KUKA KRL program: EPS_2_25362_MH2A_A_20251103083054.src

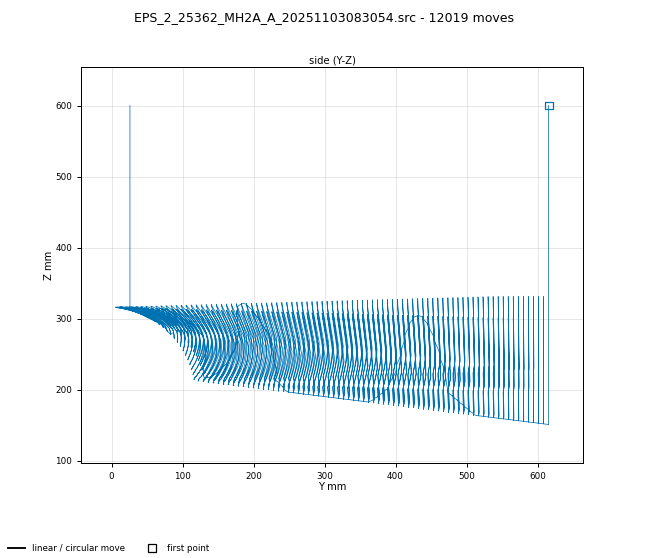
[picture p0: tool path of EPS_2_25362_MH2A_A_20251103083054.src, 12019 of 12021 moves have a stored position in this frame; points joined in program order, loops and branches not executed]
&ACCESS RVP
&REL 4
&COMMENT QRS 19112012
&PARAM EDITMASK = *
DEF PART()
EXT BAS (BAS_COMMAND :IN,REAL :IN )
INT I
BAS (#INITMOV,0 )

;KUKA QRS Post kuka4.cps  Date:22-06-2017 !

File_ID=2899

QRS_PRE_INIT()

;Init var - Until changes are made in qrs_pre_init
Outlet_Square_prg=0
Inlet_1_Square_prg=0
Inlet_2_Square_prg=0
Inlet_3_Square_prg=0
Inlet_4_Square_prg=0
Inlet_5_Square_prg=0

Outlet_1={X 0.000, Y 537.380, Z 230.500, B 0.000, E1 0.000 }
Inlet_1={X 0.000, Y 539.550, Z 200.500, B 0.000, E1 178.000 }
Outlet_1_type=201
Inlet_1_type=201
;QRS#1=Sidecore dimensions
;QRS#2=200-8" PVC SDR 35
;QRS#3=200-8" PVC SDR 35
;QRS#4=
;QRS#5=
;QRS#6=
;QRS#7=
;QRS#8=
;QRS#9=12-08 PSX
;QRS#10=12-08 PSX
;QRS#11=
;QRS#12=
;QRS#13=
;QRS#14=
;QRS#15=
;QRS#16=1220x127x610 2'
;QRS#17=EPS Height
;QRS#18=331
;QRS#19=*
;QRS#20= UPDATED VERSION 22-06-2017
;QRS#21=*
Outlet_Square=0100
Inlet_1_Square=0100
Inlet_2_Square=0
Inlet_3_Square=0
Inlet_4_Square=0
Inlet_5_Square=0
Mill_Square=1
Outlet_Square_Prg=204
Inlet_1_Square_prg=204

QRS_INIT()

$ADVANCE=5

; T1
PTP {E1 173.58,E2 173.58}
PTP {X 0,Y 615.495,A -85,B 0,C 180,E1 173.58,E2 173.58,E3 0,E4 0,E5 0,E6 0}
QRS_SPEED_INIT()
LIN {X 0,Y 615.495,Z 600,A -85,B 0,C 180,E1 173.58,E2 173.58,E3 0,E4 0,E5 0,E6 0} C_VEL
LIN {X 0,Y 615.495,Z 160.868,A -85,B 0,C 180,E1 173.58,E2 173.58} C_VEL
LIN {X 0,Y 615.495,Z 152.689,A -85,B 0,C 180,E1 173.58,E2 173.58} C_VEL
LIN {X 0,Y 615.483,Z 150.689,A -85,B 0,C 180,E1 173.393,E2 173.393} C_VEL
LIN {X 0,Y 615.483,Z 150.7,A -85,B 0,C 180,E1 170.801,E2 170.801} C_VEL
LIN {X 0,Y 615.439,Z 150.7,A -85,B 0,C 180,E1 168.138,E2 168.138} C_VEL
LIN {X 0,Y 615.491,Z 150.691,A -85,B 0,C 180,E1 165.451,E2 165.451} C_VEL
LIN {X 0,Y 615.482,Z 150.697,A -85,B 0,C 180,E1 162.729,E2 162.729} C_VEL
LIN {X 0,Y 615.477,Z 150.69,A -85,B 0,C 180,E1 159.967,E2 159.967} C_VEL
LIN {X 0,Y 615.463,Z 150.7,A -85,B 0,C 180,E1 157.154,E2 157.154} C_VEL
LIN {X 0,Y 615.457,Z 150.7,A -85,B 0,C 180,E1 154.43,E2 154.43} C_VEL
LIN {X 0,Y 615.47,Z 150.692,A -85,B 0,C 180,E1 151.546,E2 151.546} C_VEL
LIN {X 0,Y 615.484,Z 150.7,A -85,B 0,C 180,E1 148.909,E2 148.909} C_VEL
LIN {X 0,Y 615.472,Z 150.692,A -85,B 0,C 180,E1 146.463,E2 146.463} C_VEL
LIN {X 0,Y 615.451,Z 150.7,A -85,B 0,C 180,E1 143.572,E2 143.572} C_VEL
LIN {X 0,Y 615.462,Z 150.7,A -85,B 0,C 180,E1 140.936,E2 140.936} C_VEL
LIN {X 0,Y 615.493,Z 150.691,A -85,B 0,C 180,E1 138.526,E2 138.526} C_VEL
LIN {X 0,Y 615.483,Z 150.696,A -85,B 0,C 180,E1 135.849,E2 135.849} C_VEL
LIN {X 0,Y 615.463,Z 150.693,A -85,B 0,C 180,E1 133.044,E2 133.044} C_VEL
LIN {X 0,Y 615.491,Z 150.7,A -85,B 0,C 180,E1 130.603,E2 130.603} C_VEL
LIN {X 0,Y 615.445,Z 150.698,A -85,B 0,C 180,E1 128.006,E2 128.006} C_VEL
LIN {X 0,Y 615.489,Z 150.883,A -85,B 0,C 180,E1 127.239,E2 127.239} C_VEL
LIN {X 0,Y 615.484,Z 155.327,A -85,B 0,C 180,E1 124.699,E2 124.699} C_VEL
LIN {X 0,Y 615.462,Z 159.55,A -85,B 0,C 180,E1 122.326,E2 122.326} C_VEL
LIN {X 0,Y 615.495,Z 164.12,A -85,B 0,C 180,E1 119.795,E2 119.795} C_VEL
LIN {X 0,Y 615.496,Z 169.29,A -85,B 0,C 180,E1 117.045,E2 117.045} C_VEL
LIN {X 0,Y 615.488,Z 174.63,A -85,B 0,C 180,E1 114.271,E2 114.271} C_VEL
LIN {X 0,Y 615.486,Z 180.203,A -85,B 0,C 180,E1 111.431,E2 111.431} C_VEL
LIN {X 0,Y 615.475,Z 185.852,A -85,B 0,C 180,E1 108.6,E2 108.6} C_VEL
LIN {X 0,Y 615.458,Z 191.315,A -85,B 0,C 180,E1 105.905,E2 105.905} C_VEL
LIN {X 0,Y 615.497,Z 196.111,A -85,B 0,C 180,E1 103.558,E2 103.558} C_VEL
LIN {X 0,Y 615.486,Z 208.924,A -85,B 0,C 180,E1 103.285,E2 103.285} C_VEL
LIN {X 0,Y 615.445,Z 222.003,A -85,B 0,C 180,E1 102.866,E2 102.866} C_VEL
LIN {X 0,Y 615.432,Z 233.538,A -85,B 0,C 180,E1 102.363,E2 102.363} C_VEL
LIN {X 0,Y 615.477,Z 244.06,A -85,B 0,C 180,E1 101.777,E2 101.777} C_VEL
LIN {X 0,Y 615.496,Z 254.612,A -85,B 0,C 180,E1 101.041,E2 101.041} C_VEL
LIN {X 0,Y 615.498,Z 264.458,A -85,B 0,C 180,E1 100.194,E2 100.194} C_VEL
LIN {X 0,Y 615.496,Z 272.355,A -85,B 0,C 180,E1 99.364,E2 99.364} C_VEL
LIN {X 0,Y 615.497,Z 280.04,A -85,B 0,C 180,E1 98.371,E2 98.371} C_VEL
LIN {X 0,Y 615.495,Z 287.099,A -85,B 0,C 180,E1 97.215,E2 97.215} C_VEL
LIN {X 0,Y 615.496,Z 291.782,A -85,B 0,C 180,E1 96.227,E2 96.227} C_VEL
LIN {X 0,Y 615.498,Z 295.355,A -85,B 0,C 180,E1 95.241,E2 95.241} C_VEL
LIN {X 0,Y 615.496,Z 297.203,A -85,B 0,C 180,E1 94.585,E2 94.585} C_VEL
LIN {X 0,Y 615.497,Z 298.591,A -85,B 0,C 180,E1 93.929,E2 93.929} C_VEL
LIN {X 0,Y 615.495,Z 300.167,A -85,B 0,C 180,E1 92.618,E2 92.618} C_VEL
LIN {X 0,Y 615.5,Z 300.387,A -85,B 0,C 180,E1 91.963,E2 91.963} C_VEL
LIN {X 0,Y 615.495,Z 299.59,A -85,B 0,C 180,E1 90.655,E2 90.655} C_VEL
LIN {X 0,Y 615.497,Z 298.622,A -85,B 0,C 180,E1 90,E2 90} C_VEL
LIN {X 0,Y 615.494,Z 297.256,A -85,B 0,C 180,E1 89.346,E2 89.346} C_VEL
LIN {X 0,Y 615.496,Z 294.383,A -85,B 0,C 180,E1 88.365,E2 88.365} C_VEL
LIN {X 0,Y 615.498,Z 290.494,A -85,B 0,C 180,E1 87.383,E2 87.383} C_VEL
LIN {X 0,Y 615.496,Z 285.486,A -85,B 0,C 180,E1 86.4,E2 86.4} C_VEL
LIN {X 0,Y 615.498,Z 279.198,A -85,B 0,C 180,E1 85.416,E2 85.416} C_VEL
LIN {X 0,Y 615.498,Z 271.326,A -85,B 0,C 180,E1 84.431,E2 84.431} C_VEL
LIN {X 0,Y 615.498,Z 261.549,A -85,B 0,C 180,E1 83.444,E2 83.444} C_VEL
LIN {X 0,Y 615.499,Z 251.282,A -85,B 0,C 180,E1 82.621,E2 82.621} C_VEL
LIN {X 0,Y 615.454,Z 239.751,A -85,B 0,C 180,E1 81.877,E2 81.877} C_VEL
LIN {X 0,Y 615.435,Z 228.231,A -85,B 0,C 180,E1 81.298,E2 81.298} C_VEL
LIN {X 0,Y 615.465,Z 216.308,A -85,B 0,C 180,E1 80.843,E2 80.843} C_VEL
LIN {X 0,Y 615.499,Z 204.261,A -85,B 0,C 180,E1 80.512,E2 80.512} C_VEL
LIN {X 0,Y 615.487,Z 196.102,A -85,B 0,C 180,E1 80.346,E2 80.346} C_VEL
LIN {X 0,Y 615.472,Z 191.59,A -85,B 0,C 180,E1 78.14,E2 78.14} C_VEL
LIN {X 0,Y 615.467,Z 186.138,A -85,B 0,C 180,E1 75.452,E2 75.452} C_VEL
LIN {X 0,Y 615.492,Z 180.706,A -85,B 0,C 180,E1 72.731,E2 72.731} C_VEL
LIN {X 0,Y 615.478,Z 175.27,A -85,B 0,C 180,E1 69.969,E2 69.969} C_VEL
LIN {X 0,Y 615.477,Z 169.856,A -85,B 0,C 180,E1 67.157,E2 67.157} C_VEL
LIN {X 0,Y 615.493,Z 164.438,A -85,B 0,C 180,E1 64.287,E2 64.287} C_VEL
LIN {X 0,Y 615.46,Z 159.498,A -85,B 0,C 180,E1 61.556,E2 61.556} C_VEL
LIN {X 0,Y 615.49,Z 154.803,A -85,B 0,C 180,E1 58.915,E2 58.915} C_VEL
LIN {X 0,Y 615.466,Z 150.699,A -85,B 0,C 180,E1 56.47,E2 56.47} C_VEL
LIN {X 0,Y 615.43,Z 150.7,A -85,B 0,C 180,E1 54.175,E2 54.175} C_VEL
LIN {X 0,Y 615.45,Z 150.7,A -85,B 0,C 180,E1 51.933,E2 51.933} C_VEL
LIN {X 0,Y 615.489,Z 150.692,A -85,B 0,C 180,E1 49.398,E2 49.398} C_VEL
LIN {X 0,Y 615.471,Z 150.694,A -85,B 0,C 180,E1 46.758,E2 46.758} C_VEL
LIN {X 0,Y 615.477,Z 150.692,A -85,B 0,C 180,E1 44.001,E2 44.001} C_VEL
LIN {X 0,Y 615.489,Z 150.701,A -85,B 0,C 180,E1 41.1,E2 41.1} C_VEL
LIN {X 0,Y 615.453,Z 150.699,A -85,B 0,C 180,E1 38.907,E2 38.907} C_VEL
LIN {X 0,Y 615.436,Z 150.7,A -85,B 0,C 180,E1 36.429,E2 36.429} C_VEL
LIN {X 0,Y 615.463,Z 150.695,A -85,B 0,C 180,E1 33.538,E2 33.538} C_VEL
LIN {X 0,Y 615.469,Z 150.697,A -85,B 0,C 180,E1 30.921,E2 30.921} C_VEL
LIN {X 0,Y 615.485,Z 150.692,A -85,B 0,C 180,E1 28.458,E2 28.458} C_VEL
LIN {X 0,Y 615.486,Z 150.693,A -85,B 0,C 180,E1 25.716,E2 25.716} C_VEL
LIN {X 0,Y 615.483,Z 150.702,A -85,B 0,C 180,E1 23.557,E2 23.557} C_VEL
LIN {X 0,Y 615.454,Z 150.698,A -85,B 0,C 180,E1 21.433,E2 21.433} C_VEL
LIN {X 0,Y 615.428,Z 150.701,A -85,B 0,C 180,E1 19.34,E2 19.34} C_VEL
LIN {X 0,Y 615.488,Z 150.696,A -85,B 0,C 180,E1 16.447,E2 16.447} C_VEL
LIN {X 0,Y 615.457,Z 150.694,A -85,B 0,C 180,E1 13.875,E2 13.875} C_VEL
LIN {X 0,Y 615.489,Z 150.696,A -85,B 0,C 180,E1 11.193,E2 11.193} C_VEL
LIN {X 0,Y 615.49,Z 150.688,A -85,B 0,C 180,E1 8.537,E2 8.537} C_VEL
LIN {X 0,Y 615.471,Z 150.698,A -85,B 0,C 180,E1 5.899,E2 5.899} C_VEL
LIN {X 0,Y 615.456,Z 150.696,A -85,B 0,C 180,E1 3.273,E2 3.273} C_VEL
LIN {X 0,Y 615.46,Z 150.7,A -85,B 0,C 180,E1 0.654,E2 0.654} C_VEL
LIN {X 0,Y 615.444,Z 150.699,A -85,B 0,C 180,E1 -1.963,E2 -1.963} C_VEL
LIN {X 0,Y 615.493,Z 150.692,A -85,B 0,C 180,E1 -4.584,E2 -4.584} C_VEL
LIN {X 0,Y 615.478,Z 150.691,A -85,B 0,C 180,E1 -7.216,E2 -7.216} C_VEL
LIN {X 0,Y 615.474,Z 150.696,A -85,B 0,C 180,E1 -9.862,E2 -9.862} C_VEL
LIN {X 0,Y 615.49,Z 150.69,A -85,B 0,C 180,E1 -12.53,E2 -12.53} C_VEL
LIN {X 0,Y 615.445,Z 150.7,A -85,B 0,C 180,E1 -15.227,E2 -15.227} C_VEL
LIN {X 0,Y 615.429,Z 150.7,A -85,B 0,C 180,E1 -17.272,E2 -17.272} C_VEL
LIN {X 0,Y 615.49,Z 150.7,A -85,B 0,C 180,E1 -20.033,E2 -20.033} C_VEL
LIN {X 0,Y 615.467,Z 150.693,A -85,B 0,C 180,E1 -22.845,E2 -22.845} C_VEL
LIN {X 0,Y 615.481,Z 150.694,A -85,B 0,C 180,E1 -25.577,E2 -25.577} C_VEL
LIN {X 0,Y 615.49,Z 150.695,A -85,B 0,C 180,E1 -28.459,E2 -28.459} C_VEL
LIN {X 0,Y 615.448,Z 150.697,A -85,B 0,C 180,E1 -31.088,E2 -31.088} C_VEL
LIN {X 0,Y 615.458,Z 150.699,A -85,B 0,C 180,E1 -33.537,E2 -33.537} C_VEL
LIN {X 0,Y 615.488,Z 150.697,A -85,B 0,C 180,E1 -35.84,E2 -35.84} C_VEL
LIN {X 0,Y 615.467,Z 150.692,A -85,B 0,C 180,E1 -38.07,E2 -38.07} C_VEL
LIN {X 0,Y 615.473,Z 150.698,A -85,B 0,C 180,E1 -40.608,E2 -40.608} C_VEL
LIN {X 0,Y 615.483,Z 150.689,A -85,B 0,C 180,E1 -43.245,E2 -43.245} C_VEL
LIN {X 0,Y 615.485,Z 150.699,A -85,B 0,C 180,E1 -46.003,E2 -46.003} C_VEL
LIN {X 0,Y 615.449,Z 150.696,A -85,B 0,C 180,E1 -48.527,E2 -48.527} C_VEL
LIN {X 0,Y 615.472,Z 150.698,A -85,B 0,C 180,E1 -51.098,E2 -51.098} C_VEL
LIN {X 0,Y 615.459,Z 150.697,A -85,B 0,C 180,E1 -53.577,E2 -53.577} C_VEL
LIN {X 0,Y 615.468,Z 150.796,A -85,B 0,C 180,E1 -54.587,E2 -54.587} C_VEL
LIN {X 0,Y 615.486,Z 157.959,A -85,B 0,C 180,E1 -57.157,E2 -57.157} C_VEL
LIN {X 0,Y 615.486,Z 165.755,A -85,B 0,C 180,E1 -59.843,E2 -59.843} C_VEL
LIN {X 0,Y 615.467,Z 173.553,A -85,B 0,C 180,E1 -62.456,E2 -62.456} C_VEL
LIN {X 0,Y 615.492,Z 181.317,A -85,B 0,C 180,E1 -65.011,E2 -65.011} C_VEL
LIN {X 0,Y 615.461,Z 190.18,A -85,B 0,C 180,E1 -67.865,E2 -67.865} C_VEL
LIN {X 0,Y 615.466,Z 197.941,A -85,B 0,C 180,E1 -70.316,E2 -70.316} C_VEL
LIN {X 0,Y 615.487,Z 206.786,A -85,B 0,C 180,E1 -73.073,E2 -73.073} C_VEL
LIN {X 0,Y 615.439,Z 215.576,A -85,B 0,C 180,E1 -75.766,E2 -75.766} C_VEL
LIN {X 0,Y 615.489,Z 224.141,A -85,B 0,C 180,E1 -78.37,E2 -78.37} C_VEL
LIN {X 0,Y 615.492,Z 236.12,A -85,B 0,C 180,E1 -78.6,E2 -78.6} C_VEL
LIN {X 0,Y 615.45,Z 248.862,A -85,B 0,C 180,E1 -78.972,E2 -78.972} C_VEL
LIN {X 0,Y 615.429,Z 261.057,A -85,B 0,C 180,E1 -79.473,E2 -79.473} C_VEL
LIN {X 0,Y 615.464,Z 272.005,A -85,B 0,C 180,E1 -80.056,E2 -80.056} C_VEL
LIN {X 0,Y 615.499,Z 283.182,A -85,B 0,C 180,E1 -80.803,E2 -80.803} C_VEL
LIN {X 0,Y 615.498,Z 293.056,A -85,B 0,C 180,E1 -81.63,E2 -81.63} C_VEL
LIN {X 0,Y 615.498,Z 302.615,A -85,B 0,C 180,E1 -82.621,E2 -82.621} C_VEL
LIN {X 0,Y 615.496,Z 310.209,A -85,B 0,C 180,E1 -83.609,E2 -83.609} C_VEL
LIN {X 0,Y 615.498,Z 317.209,A -85,B 0,C 180,E1 -84.76,E2 -84.76} C_VEL
LIN {X 0,Y 615.493,Z 321.855,A -85,B 0,C 180,E1 -85.744,E2 -85.744} C_VEL
LIN {X 0,Y 615.494,Z 325.401,A -85,B 0,C 180,E1 -86.728,E2 -86.728} C_VEL
LIN {X 0,Y 615.497,Z 327.234,A -85,B 0,C 180,E1 -87.383,E2 -87.383} C_VEL
LIN {X 0,Y 615.5,Z 328.608,A -85,B 0,C 180,E1 -88.038,E2 -88.038} C_VEL
LIN {X 0,Y 615.496,Z 330.174,A -85,B 0,C 180,E1 -89.346,E2 -89.346} C_VEL
LIN {X 0,Y 615.494,Z 330.389,A -85,B 0,C 180,E1 -90,E2 -90} C_VEL
LIN {X 0,Y 615.495,Z 329.58,A -85,B 0,C 180,E1 -91.309,E2 -91.309} C_VEL
LIN {X 0,Y 615.5,Z 328.607,A -85,B 0,C 180,E1 -91.963,E2 -91.963} C_VEL
LIN {X 0,Y 615.497,Z 327.232,A -85,B 0,C 180,E1 -92.618,E2 -92.618} C_VEL
LIN {X 0,Y 615.496,Z 324.349,A -85,B 0,C 180,E1 -93.601,E2 -93.601} C_VEL
LIN {X 0,Y 615.498,Z 320.441,A -85,B 0,C 180,E1 -94.585,E2 -94.585} C_VEL
LIN {X 0,Y 615.499,Z 315.405,A -85,B 0,C 180,E1 -95.57,E2 -95.57} C_VEL
LIN {X 0,Y 615.497,Z 308.869,A -85,B 0,C 180,E1 -96.583,E2 -96.583} C_VEL
LIN {X 0,Y 615.498,Z 301.134,A -85,B 0,C 180,E1 -97.545,E2 -97.545} C_VEL
LIN {X 0,Y 615.498,Z 293.047,A -85,B 0,C 180,E1 -98.371,E2 -98.371} C_VEL
LIN {X 0,Y 615.499,Z 283.17,A -85,B 0,C 180,E1 -99.198,E2 -99.198} C_VEL
LIN {X 0,Y 615.463,Z 271.99,A -85,B 0,C 180,E1 -99.945,E2 -99.945} C_VEL
LIN {X 0,Y 615.429,Z 261.039,A -85,B 0,C 180,E1 -100.528,E2 -100.528} C_VEL
LIN {X 0,Y 615.451,Z 248.849,A -85,B 0,C 180,E1 -101.028,E2 -101.028} C_VEL
LIN {X 0,Y 615.492,Z 236.081,A -85,B 0,C 180,E1 -101.401,E2 -101.401} C_VEL
LIN {X 0,Y 615.489,Z 224.138,A -85,B 0,C 180,E1 -101.631,E2 -101.631} C_VEL
LIN {X 0,Y 615.44,Z 215.574,A -85,B 0,C 180,E1 -104.235,E2 -104.235} C_VEL
LIN {X 0,Y 615.487,Z 206.783,A -85,B 0,C 180,E1 -106.927,E2 -106.927} C_VEL
LIN {X 0,Y 615.466,Z 197.938,A -85,B 0,C 180,E1 -109.685,E2 -109.685} C_VEL
LIN {X 0,Y 615.471,Z 189.53,A -85,B 0,C 180,E1 -112.342,E2 -112.342} C_VEL
LIN {X 0,Y 615.492,Z 181.314,A -85,B 0,C 180,E1 -114.99,E2 -114.99} C_VEL
LIN {X 0,Y 615.468,Z 173.55,A -85,B 0,C 180,E1 -117.545,E2 -117.545} C_VEL
LIN {X 0,Y 615.486,Z 165.751,A -85,B 0,C 180,E1 -120.158,E2 -120.158} C_VEL
LIN {X 0,Y 615.486,Z 157.955,A -85,B 0,C 180,E1 -122.844,E2 -122.844} C_VEL
LIN {X 0,Y 615.463,Z 150.7,A -85,B 0,C 180,E1 -125.464,E2 -125.464} C_VEL
LIN {X 0,Y 615.444,Z 150.701,A -85,B 0,C 180,E1 -128.069,E2 -128.069} C_VEL
LIN {X 0,Y 615.489,Z 150.692,A -85,B 0,C 180,E1 -130.603,E2 -130.603} C_VEL
LIN {X 0,Y 615.479,Z 150.695,A -85,B 0,C 180,E1 -133.242,E2 -133.242} C_VEL
LIN {X 0,Y 615.469,Z 150.692,A -85,B 0,C 180,E1 -136.001,E2 -136.001} C_VEL
LIN {X 0,Y 615.463,Z 150.7,A -85,B 0,C 180,E1 -138.904,E2 -138.904} C_VEL
LIN {X 0,Y 615.436,Z 150.7,A -85,B 0,C 180,E1 -141.092,E2 -141.092} C_VEL
LIN {X 0,Y 615.482,Z 150.701,A -85,B 0,C 180,E1 -143.575,E2 -143.575} C_VEL
LIN {X 0,Y 615.482,Z 150.691,A -85,B 0,C 180,E1 -146.461,E2 -146.461} C_VEL
LIN {X 0,Y 615.469,Z 150.697,A -85,B 0,C 180,E1 -149.079,E2 -149.079} C_VEL
LIN {X 0,Y 615.459,Z 150.697,A -85,B 0,C 180,E1 -151.548,E2 -151.548} C_VEL
LIN {X 0,Y 615.447,Z 150.698,A -85,B 0,C 180,E1 -154.431,E2 -154.431} C_VEL
LIN {X 0,Y 615.46,Z 150.695,A -85,B 0,C 180,E1 -156.443,E2 -156.443} C_VEL
LIN {X 0,Y 615.481,Z 150.697,A -85,B 0,C 180,E1 -158.568,E2 -158.568} C_VEL
LIN {X 0,Y 615.481,Z 150.689,A -85,B 0,C 180,E1 -161.386,E2 -161.386} C_VEL
LIN {X 0,Y 615.469,Z 150.7,A -85,B 0,C 180,E1 -164.094,E2 -164.094} C_VEL
LIN {X 0,Y 615.439,Z 150.7,A -85,B 0,C 180,E1 -166.125,E2 -166.125} C_VEL
LIN {X 0,Y 615.483,Z 150.701,A -85,B 0,C 180,E1 -168.807,E2 -168.807} C_VEL
LIN {X 0,Y 615.487,Z 150.688,A -85,B 0,C 180,E1 -171.463,E2 -171.463} C_VEL
LIN {X 0,Y 615.484,Z 150.699,A -85,B 0,C 180,E1 -174.102,E2 -174.102} C_VEL
LIN {X 0,Y 615.458,Z 150.696,A -85,B 0,C 180,E1 -176.727,E2 -176.727} C_VEL
LIN {X 0,Y 615.461,Z 150.699,A -85,B 0,C 180,E1 -179.346,E2 -179.346} C_VEL
LIN {X 0,Y 615.463,Z 150.698,A -85,B 0,C 180,E1 -181.963,E2 -181.963} C_VEL
LIN {X 0,Y 615.487,Z 150.69,A -85,B 0,C 180,E1 -184.585,E2 -184.585} C_VEL
LIN {X 0,Y 615.483,Z 150.689,A -85,B 0,C 180,E1 -186.607,E2 -186.607} C_VEL
LIN {X 0,Y 614.815,Z 150.844,A -85,B 0,C 180,E1 -187.153,E2 -187.153} C_VEL
LIN {X 0,Y 611.982,Z 151.251,A -85,B 0,C 180,E1 -188.039,E2 -188.039} C_VEL
LIN {X 0,Y 609.582,Z 151.565,A -85,B 0,C 180,E1 -188.751,E2 -188.751} C_VEL
LIN {X 0,Y 608.534,Z 151.685,A -85,B 0,C 180,E1 -189.301,E2 -189.301} C_VEL
LIN {X 0,Y 608.44,Z 151.694,A -85,B 0,C 180,E1 -189.487,E2 -189.487} C_VEL
LIN {X 0,Y 608.426,Z 151.695,A -85,B 0,C 180,E1 -192.001,E2 -192.001} C_VEL
LIN {X 0,Y 608.467,Z 151.689,A -85,B 0,C 180,E1 -194.721,E2 -194.721} C_VEL
LIN {X 0,Y 608.463,Z 151.689,A -85,B 0,C 180,E1 -196.784,E2 -196.784} C_VEL
LIN {X 0,Y 608.446,Z 151.694,A -85,B 0,C 180,E1 -199.571,E2 -199.571} C_VEL
LIN {X 0,Y 608.465,Z 151.696,A -85,B 0,C 180,E1 -202.486,E2 -202.486} C_VEL
LIN {X 0,Y 608.428,Z 151.696,A -85,B 0,C 180,E1 -204.572,E2 -204.572} C_VEL
LIN {X 0,Y 608.451,Z 151.693,A -85,B 0,C 180,E1 -207.209,E2 -207.209} C_VEL
LIN {X 0,Y 608.468,Z 151.689,A -85,B 0,C 180,E1 -209.978,E2 -209.978} C_VEL
LIN {X 0,Y 608.445,Z 151.696,A -85,B 0,C 180,E1 -212.881,E2 -212.881} C_VEL
LIN {X 0,Y 608.423,Z 151.694,A -85,B 0,C 180,E1 -215.279,E2 -215.279} C_VEL
LIN {X 0,Y 608.441,Z 151.693,A -85,B 0,C 180,E1 -218.242,E2 -218.242} C_VEL
LIN {X 0,Y 608.427,Z 151.694,A -85,B 0,C 180,E1 -220.33,E2 -220.33} C_VEL
LIN {X 0,Y 608.451,Z 151.695,A -85,B 0,C 180,E1 -222.961,E2 -222.961} C_VEL
LIN {X 0,Y 608.455,Z 151.693,A -85,B 0,C 180,E1 -225.737,E2 -225.737} C_VEL
LIN {X 0,Y 608.462,Z 151.695,A -85,B 0,C 180,E1 -227.942,E2 -227.942} C_VEL
LIN {X 0,Y 608.421,Z 151.696,A -85,B 0,C 180,E1 -230.709,E2 -230.709} C_VEL
LIN {X 0,Y 608.41,Z 151.696,A -85,B 0,C 180,E1 -232.252,E2 -232.252} C_VEL
LIN {X 0,Y 608.481,Z 152.01,A -85,B 0,C 180,E1 -232.841,E2 -232.841} C_VEL
LIN {X 0,Y 608.435,Z 156.696,A -85,B 0,C 180,E1 -235.531,E2 -235.531} C_VEL
LIN {X 0,Y 608.422,Z 160.891,A -85,B 0,C 180,E1 -237.905,E2 -237.905} C_VEL
LIN {X 0,Y 608.46,Z 165.046,A -85,B 0,C 180,E1 -240.222,E2 -240.222} C_VEL
LIN {X 0,Y 608.429,Z 170.654,A -85,B 0,C 180,E1 -243.226,E2 -243.226} C_VEL
LIN {X 0,Y 608.451,Z 175.687,A -85,B 0,C 180,E1 -245.854,E2 -245.854} C_VEL
LIN {X 0,Y 608.414,Z 180.475,A -85,B 0,C 180,E1 -248.308,E2 -248.308} C_VEL
LIN {X 0,Y 608.431,Z 186.073,A -85,B 0,C 180,E1 -251.131,E2 -251.131} C_VEL
LIN {X 0,Y 608.415,Z 191.659,A -85,B 0,C 180,E1 -253.906,E2 -253.906} C_VEL
LIN {X 0,Y 608.445,Z 196.631,A -85,B 0,C 180,E1 -256.314,E2 -256.314} C_VEL
LIN {X 0,Y 608.535,Z 209.722,A -85,B 0,C 180,E1 -256.603,E2 -256.603} C_VEL
LIN {X 0,Y 608.487,Z 222.634,A -85,B 0,C 180,E1 -257.027,E2 -257.027} C_VEL
LIN {X 0,Y 608.438,Z 234.898,A -85,B 0,C 180,E1 -257.577,E2 -257.577} C_VEL
LIN {X 0,Y 608.49,Z 246.48,A -85,B 0,C 180,E1 -258.255,E2 -258.255} C_VEL
LIN {X 0,Y 608.48,Z 257.238,A -85,B 0,C 180,E1 -259.042,E2 -259.042} C_VEL
LIN {X 0,Y 608.482,Z 266.246,A -85,B 0,C 180,E1 -259.855,E2 -259.855} C_VEL
LIN {X 0,Y 608.47,Z 275.279,A -85,B 0,C 180,E1 -260.862,E2 -260.862} C_VEL
LIN {X 0,Y 608.463,Z 282.55,A -85,B 0,C 180,E1 -261.866,E2 -261.866} C_VEL
LIN {X 0,Y 608.445,Z 287.448,A -85,B 0,C 180,E1 -262.7,E2 -262.7} C_VEL
LIN {X 0,Y 608.452,Z 291.911,A -85,B 0,C 180,E1 -263.632,E2 -263.632} C_VEL
LIN {X 0,Y 608.442,Z 295.84,A -85,B 0,C 180,E1 -264.698,E2 -264.698} C_VEL
LIN {X 0,Y 608.429,Z 297.718,A -85,B 0,C 180,E1 -265.362,E2 -265.362} C_VEL
LIN {X 0,Y 608.434,Z 299.146,A -85,B 0,C 180,E1 -266.026,E2 -266.026} C_VEL
LIN {X 0,Y 608.421,Z 300.761,A -85,B 0,C 180,E1 -267.351,E2 -267.351} C_VEL
LIN {X 0,Y 608.445,Z 300.998,A -85,B 0,C 180,E1 -268.014,E2 -268.014} C_VEL
LIN {X 0,Y 608.447,Z 300.805,A -85,B 0,C 180,E1 -268.676,E2 -268.676} C_VEL
LIN {X 0,Y 608.437,Z 299.253,A -85,B 0,C 180,E1 -270,E2 -270} C_VEL
LIN {X 0,Y 608.437,Z 297.888,A -85,B 0,C 180,E1 -270.661,E2 -270.661} C_VEL
LIN {X 0,Y 608.44,Z 295.004,A -85,B 0,C 180,E1 -271.654,E2 -271.654} C_VEL
LIN {X 0,Y 608.432,Z 291.101,A -85,B 0,C 180,E1 -272.648,E2 -272.648} C_VEL
LIN {X 0,Y 608.449,Z 286.073,A -85,B 0,C 180,E1 -273.642,E2 -273.642} C_VEL
LIN {X 0,Y 608.465,Z 279.766,A -85,B 0,C 180,E1 -274.637,E2 -274.637} C_VEL
LIN {X 0,Y 608.47,Z 271.876,A -85,B 0,C 180,E1 -275.633,E2 -275.633} C_VEL
LIN {X 0,Y 608.484,Z 262.08,A -85,B 0,C 180,E1 -276.632,E2 -276.632} C_VEL
LIN {X 0,Y 608.479,Z 251.829,A -85,B 0,C 180,E1 -277.465,E2 -277.465} C_VEL
LIN {X 0,Y 608.471,Z 240.31,A -85,B 0,C 180,E1 -278.217,E2 -278.217} C_VEL
LIN {X 0,Y 608.467,Z 228.903,A -85,B 0,C 180,E1 -278.802,E2 -278.802} C_VEL
LIN {X 0,Y 608.494,Z 217.135,A -85,B 0,C 180,E1 -279.262,E2 -279.262} C_VEL
LIN {X 0,Y 608.557,Z 203.56,A -85,B 0,C 180,E1 -279.639,E2 -279.639} C_VEL
LIN {X 0,Y 608.419,Z 196.539,A -85,B 0,C 180,E1 -279.788,E2 -279.788} C_VEL
LIN {X 0,Y 608.416,Z 192.034,A -85,B 0,C 180,E1 -281.999,E2 -281.999} C_VEL
LIN {X 0,Y 608.405,Z 186.552,A -85,B 0,C 180,E1 -284.721,E2 -284.721} C_VEL
LIN {X 0,Y 608.433,Z 181.079,A -85,B 0,C 180,E1 -287.475,E2 -287.475} C_VEL
LIN {X 0,Y 608.425,Z 175.616,A -85,B 0,C 180,E1 -290.273,E2 -290.273} C_VEL
LIN {X 0,Y 608.441,Z 171.399,A -85,B 0,C 180,E1 -292.471,E2 -292.471} C_VEL
LIN {X 0,Y 608.45,Z 167.441,A -85,B 0,C 180,E1 -294.569,E2 -294.569} C_VEL
LIN {X 0,Y 608.463,Z 162.632,A -85,B 0,C 180,E1 -297.203,E2 -297.203} C_VEL
LIN {X 0,Y 608.432,Z 157.741,A -85,B 0,C 180,E1 -299.965,E2 -299.965} C_VEL
LIN {X 0,Y 608.446,Z 152.643,A -85,B 0,C 180,E1 -302.877,E2 -302.877} C_VEL
LIN {X 0,Y 608.434,Z 151.694,A -85,B 0,C 180,E1 -303.729,E2 -303.729} C_VEL
LIN {X 0,Y 608.421,Z 151.694,A -85,B 0,C 180,E1 -306.09,E2 -306.09} C_VEL
LIN {X 0,Y 608.45,Z 151.697,A -85,B 0,C 180,E1 -308.586,E2 -308.586} C_VEL
LIN {X 0,Y 608.439,Z 151.692,A -85,B 0,C 180,E1 -311.339,E2 -311.339} C_VEL
LIN {X 0,Y 608.451,Z 151.691,A -85,B 0,C 180,E1 -314.263,E2 -314.263} C_VEL
LIN {X 0,Y 608.452,Z 151.696,A -85,B 0,C 180,E1 -317.04,E2 -317.04} C_VEL
LIN {X 0,Y 608.428,Z 151.693,A -85,B 0,C 180,E1 -319.694,E2 -319.694} C_VEL
LIN {X 0,Y 608.447,Z 151.696,A -85,B 0,C 180,E1 -322.252,E2 -322.252} C_VEL
LIN {X 0,Y 608.413,Z 151.696,A -85,B 0,C 180,E1 -324.72,E2 -324.72} C_VEL
LIN {X 0,Y 608.454,Z 151.695,A -85,B 0,C 180,E1 -327.471,E2 -327.471} C_VEL
LIN {X 0,Y 608.465,Z 151.688,A -85,B 0,C 180,E1 -330.22,E2 -330.22} C_VEL
LIN {X 0,Y 608.475,Z 151.694,A -85,B 0,C 180,E1 -332.784,E2 -332.784} C_VEL
LIN {X 0,Y 608.442,Z 151.691,A -85,B 0,C 180,E1 -335.428,E2 -335.428} C_VEL
LIN {X 0,Y 608.45,Z 151.696,A -85,B 0,C 180,E1 -338.307,E2 -338.307} C_VEL
LIN {X 0,Y 608.412,Z 151.696,A -85,B 0,C 180,E1 -340.428,E2 -340.428} C_VEL
LIN {X 0,Y 608.487,Z 151.692,A -85,B 0,C 180,E1 -343.449,E2 -343.449} C_VEL
LIN {X 0,Y 608.433,Z 151.692,A -85,B 0,C 180,E1 -345.978,E2 -345.978} C_VEL
LIN {X 0,Y 608.462,Z 151.696,A -85,B 0,C 180,E1 -348.676,E2 -348.676} C_VEL
LIN {X 0,Y 608.454,Z 151.69,A -85,B 0,C 180,E1 -351.364,E2 -351.364} C_VEL
LIN {X 0,Y 608.468,Z 151.693,A -85,B 0,C 180,E1 -354.033,E2 -354.033} C_VEL
LIN {X 0,Y 608.448,Z 151.691,A -85,B 0,C 180,E1 -356.689,E2 -356.689} C_VEL
LIN {X 0,Y 608.452,Z 151.694,A -85,B 0,C 180,E1 -359.338,E2 -359.338} C_VEL
LIN {X 0,Y 608.416,Z 151.696,A -85,B 0,C 180,E1 -361.986,E2 -361.986} C_VEL
LIN {X 0,Y 608.459,Z 151.692,A -85,B 0,C 180,E1 -364.637,E2 -364.637} C_VEL
LIN {X 0,Y 608.464,Z 151.69,A -85,B 0,C 180,E1 -367.299,E2 -367.299} C_VEL
LIN {X 0,Y 608.444,Z 151.693,A -85,B 0,C 180,E1 -369.977,E2 -369.977} C_VEL
LIN {X 0,Y 608.471,Z 151.691,A -85,B 0,C 180,E1 -372.677,E2 -372.677} C_VEL
LIN {X 0,Y 608.428,Z 151.693,A -85,B 0,C 180,E1 -375.407,E2 -375.407} C_VEL
LIN {X 0,Y 608.427,Z 151.701,A -85,B 0,C 180,E1 -378.172,E2 -378.172} C_VEL
LIN {X 0,Y 608.431,Z 151.693,A -85,B 0,C 180,E1 -380.982,E2 -380.982} C_VEL
LIN {X 0,Y 608.437,Z 151.695,A -85,B 0,C 180,E1 -383.125,E2 -383.125} C_VEL
LIN {X 0,Y 608.459,Z 151.69,A -85,B 0,C 180,E1 -385.728,E2 -385.728} C_VEL
LIN {X 0,Y 608.471,Z 151.695,A -85,B 0,C 180,E1 -388.628,E2 -388.628} C_VEL
LIN {X 0,Y 608.445,Z 151.691,A -85,B 0,C 180,E1 -391.318,E2 -391.318} C_VEL
LIN {X 0,Y 608.45,Z 151.696,A -85,B 0,C 180,E1 -393.739,E2 -393.739} C_VEL
LIN {X 0,Y 608.45,Z 151.692,A -85,B 0,C 180,E1 -396.092,E2 -396.092} C_VEL
LIN {X 0,Y 608.453,Z 151.691,A -85,B 0,C 180,E1 -398.589,E2 -398.589} C_VEL
LIN {X 0,Y 608.464,Z 151.69,A -85,B 0,C 180,E1 -401.348,E2 -401.348} C_VEL
LIN {X 0,Y 608.452,Z 151.696,A -85,B 0,C 180,E1 -404.268,E2 -404.268} C_VEL
LIN {X 0,Y 608.435,Z 151.692,A -85,B 0,C 180,E1 -407.043,E2 -407.043} C_VEL
LIN {X 0,Y 608.439,Z 151.699,A -85,B 0,C 180,E1 -409.7,E2 -409.7} C_VEL
LIN {X 0,Y 608.457,Z 151.694,A -85,B 0,C 180,E1 -412.843,E2 -412.843} C_VEL
LIN {X 0,Y 608.44,Z 151.77,A -85,B 0,C 180,E1 -414.472,E2 -414.472} C_VEL
LIN {X 0,Y 608.492,Z 159.088,A -85,B 0,C 180,E1 -417.126,E2 -417.126} C_VEL
LIN {X 0,Y 608.487,Z 167.446,A -85,B 0,C 180,E1 -420.026,E2 -420.026} C_VEL
LIN {X 0,Y 608.48,Z 175.676,A -85,B 0,C 180,E1 -422.793,E2 -422.793} C_VEL
LIN {X 0,Y 608.462,Z 183.664,A -85,B 0,C 180,E1 -425.432,E2 -425.432} C_VEL
LIN {X 0,Y 608.424,Z 191.455,A -85,B 0,C 180,E1 -427.952,E2 -427.952} C_VEL
LIN {X 0,Y 608.447,Z 199.245,A -85,B 0,C 180,E1 -430.431,E2 -430.431} C_VEL
LIN {X 0,Y 608.441,Z 208.149,A -85,B 0,C 180,E1 -433.217,E2 -433.217} C_VEL
LIN {X 0,Y 608.42,Z 217.053,A -85,B 0,C 180,E1 -435.963,E2 -435.963} C_VEL
LIN {X 0,Y 608.427,Z 224.496,A -85,B 0,C 180,E1 -438.233,E2 -438.233} C_VEL
LIN {X 0,Y 608.552,Z 237.981,A -85,B 0,C 180,E1 -438.51,E2 -438.51} C_VEL
LIN {X 0,Y 608.481,Z 250.05,A -85,B 0,C 180,E1 -438.885,E2 -438.885} C_VEL
LIN {X 0,Y 608.459,Z 262.947,A -85,B 0,C 180,E1 -439.435,E2 -439.435} C_VEL
LIN {X 0,Y 608.463,Z 273.599,A -85,B 0,C 180,E1 -440.024,E2 -440.024} C_VEL
LIN {X 0,Y 608.483,Z 284.489,A -85,B 0,C 180,E1 -440.779,E2 -440.779} C_VEL
LIN {X 0,Y 608.475,Z 295.123,A -85,B 0,C 180,E1 -441.7,E2 -441.7} C_VEL
LIN {X 0,Y 608.47,Z 302.969,A -85,B 0,C 180,E1 -442.535,E2 -442.535} C_VEL
LIN {X 0,Y 608.46,Z 310.29,A -85,B 0,C 180,E1 -443.485,E2 -443.485} C_VEL
LIN {X 0,Y 608.45,Z 315.871,A -85,B 0,C 180,E1 -444.366,E2 -444.366} C_VEL
LIN {X 0,Y 608.432,Z 320.953,A -85,B 0,C 180,E1 -445.363,E2 -445.363} C_VEL
LIN {X 0,Y 608.449,Z 324.898,A -85,B 0,C 180,E1 -446.358,E2 -446.358} C_VEL
LIN {X 0,Y 608.425,Z 327.811,A -85,B 0,C 180,E1 -447.352,E2 -447.352} C_VEL
LIN {X 0,Y 608.444,Z 329.202,A -85,B 0,C 180,E1 -448.015,E2 -448.015} C_VEL
LIN {X 0,Y 608.438,Z 330.784,A -85,B 0,C 180,E1 -449.339,E2 -449.339} C_VEL
LIN {X 0,Y 608.434,Z 331,A -85,B 0,C 180,E1 -450,E2 -450} C_VEL
LIN {X 0,Y 608.448,Z 330.183,A -85,B 0,C 180,E1 -451.324,E2 -451.324} C_VEL
LIN {X 0,Y 608.444,Z 329.201,A -85,B 0,C 180,E1 -451.986,E2 -451.986} C_VEL
LIN {X 0,Y 608.425,Z 327.809,A -85,B 0,C 180,E1 -452.649,E2 -452.649} C_VEL
LIN {X 0,Y 608.449,Z 324.896,A -85,B 0,C 180,E1 -453.643,E2 -453.643} C_VEL
LIN {X 0,Y 608.432,Z 320.949,A -85,B 0,C 180,E1 -454.638,E2 -454.638} C_VEL
LIN {X 0,Y 608.438,Z 314.876,A -85,B 0,C 180,E1 -455.801,E2 -455.801} C_VEL
LIN {X 0,Y 608.462,Z 308.235,A -85,B 0,C 180,E1 -456.799,E2 -456.799} C_VEL
LIN {X 0,Y 608.456,Z 299.99,A -85,B 0,C 180,E1 -457.8,E2 -457.8} C_VEL
LIN {X 0,Y 608.472,Z 291.538,A -85,B 0,C 180,E1 -458.636,E2 -458.636} C_VEL
LIN {X 0,Y 608.48,Z 281.094,A -85,B 0,C 180,E1 -459.473,E2 -459.473} C_VEL
LIN {X 0,Y 608.457,Z 270.761,A -85,B 0,C 180,E1 -460.145,E2 -460.145} C_VEL
LIN {X 0,Y 608.456,Z 259.914,A -85,B 0,C 180,E1 -460.711,E2 -460.711} C_VEL
LIN {X 0,Y 608.487,Z 248.136,A -85,B 0,C 180,E1 -461.185,E2 -461.185} C_VEL
LIN {X 0,Y 608.545,Z 235.283,A -85,B 0,C 180,E1 -461.554,E2 -461.554} C_VEL
LIN {X 0,Y 608.427,Z 224.493,A -85,B 0,C 180,E1 -461.768,E2 -461.768} C_VEL
LIN {X 0,Y 608.387,Z 215.937,A -85,B 0,C 180,E1 -464.38,E2 -464.38} C_VEL
LIN {X 0,Y 608.442,Z 208.146,A -85,B 0,C 180,E1 -466.784,E2 -466.784} C_VEL
LIN {X 0,Y 608.447,Z 199.242,A -85,B 0,C 180,E1 -469.57,E2 -469.57} C_VEL
LIN {X 0,Y 608.424,Z 191.452,A -85,B 0,C 180,E1 -472.049,E2 -472.049} C_VEL
LIN {X 0,Y 608.462,Z 183.661,A -85,B 0,C 180,E1 -474.569,E2 -474.569} C_VEL
LIN {X 0,Y 608.481,Z 175.675,A -85,B 0,C 180,E1 -477.207,E2 -477.207} C_VEL
LIN {X 0,Y 608.488,Z 167.435,A -85,B 0,C 180,E1 -479.974,E2 -479.974} C_VEL
LIN {X 0,Y 608.494,Z 159.083,A -85,B 0,C 180,E1 -482.875,E2 -482.875} C_VEL
LIN {X 0,Y 608.427,Z 151.698,A -85,B 0,C 180,E1 -485.556,E2 -485.556} C_VEL
LIN {X 0,Y 608.434,Z 151.696,A -85,B 0,C 180,E1 -488.236,E2 -488.236} C_VEL
LIN {X 0,Y 608.436,Z 151.693,A -85,B 0,C 180,E1 -491.175,E2 -491.175} C_VEL
LIN {X 0,Y 608.462,Z 151.693,A -85,B 0,C 180,E1 -493.867,E2 -493.867} C_VEL
LIN {X 0,Y 608.479,Z 151.691,A -85,B 0,C 180,E1 -496.687,E2 -496.687} C_VEL
LIN {X 0,Y 608.439,Z 151.697,A -85,B 0,C 180,E1 -498.822,E2 -498.822} C_VEL
LIN {X 0,Y 608.409,Z 151.697,A -85,B 0,C 180,E1 -501.407,E2 -501.407} C_VEL
LIN {X 0,Y 608.464,Z 151.692,A -85,B 0,C 180,E1 -503.947,E2 -503.947} C_VEL
LIN {X 0,Y 608.461,Z 151.69,A -85,B 0,C 180,E1 -506.329,E2 -506.329} C_VEL
LIN {X 0,Y 608.46,Z 151.697,A -85,B 0,C 180,E1 -508.724,E2 -508.724} C_VEL
LIN {X 0,Y 608.441,Z 151.692,A -85,B 0,C 180,E1 -511.379,E2 -511.379} C_VEL
LIN {X 0,Y 608.438,Z 151.693,A -85,B 0,C 180,E1 -514.278,E2 -514.278} C_VEL
LIN {X 0,Y 608.438,Z 151.696,A -85,B 0,C 180,E1 -516.876,E2 -516.876} C_VEL
LIN {X 0,Y 608.459,Z 151.691,A -85,B 0,C 180,E1 -519.314,E2 -519.314} C_VEL
LIN {X 0,Y 608.453,Z 151.693,A -85,B 0,C 180,E1 -521.828,E2 -521.828} C_VEL
LIN {X 0,Y 608.433,Z 151.693,A -85,B 0,C 180,E1 -524.593,E2 -524.593} C_VEL
LIN {X 0,Y 608.465,Z 151.695,A -85,B 0,C 180,E1 -527.323,E2 -527.323} C_VEL
LIN {X 0,Y 608.439,Z 151.693,A -85,B 0,C 180,E1 -530.023,E2 -530.023} C_VEL
LIN {X 0,Y 608.468,Z 151.69,A -85,B 0,C 180,E1 -532.701,E2 -532.701} C_VEL
LIN {X 0,Y 608.461,Z 151.693,A -85,B 0,C 180,E1 -535.363,E2 -535.363} C_VEL
LIN {X 0,Y 608.407,Z 151.696,A -85,B 0,C 180,E1 -538.014,E2 -538.014} C_VEL
LIN {X 0,Y 608.477,Z 151.695,A -85,B 0,C 180,E1 -540.662,E2 -540.662} C_VEL
LIN {X 0,Y 608.465,Z 151.689,A -85,B 0,C 180,E1 -543.311,E2 -543.311} C_VEL
LIN {X 0,Y 608.48,Z 151.691,A -85,B 0,C 180,E1 -545.967,E2 -545.967} C_VEL
LIN {X 0,Y 608.449,Z 151.692,A -85,B 0,C 180,E1 -548.636,E2 -548.636} C_VEL
LIN {X 0,Y 608.44,Z 151.694,A -85,B 0,C 180,E1 -549.487,E2 -549.487} C_VEL
LIN {X 0,Y 607.746,Z 151.779,A -85,B 0,C 180,E1 -550.04,E2 -550.04} C_VEL
LIN {X 0,Y 604.882,Z 152.141,A -85,B 0,C 180,E1 -550.937,E2 -550.937} C_VEL
LIN {X 0,Y 602.484,Z 152.439,A -85,B 0,C 180,E1 -551.658,E2 -551.658} C_VEL
LIN {X 0,Y 601.463,Z 152.565,A -85,B 0,C 180,E1 -552.215,E2 -552.215} C_VEL
LIN {X 0,Y 601.384,Z 152.573,A -85,B 0,C 180,E1 -552.403,E2 -552.403} C_VEL
LIN {X 0,Y 601.416,Z 152.567,A -85,B 0,C 180,E1 -554.898,E2 -554.898} C_VEL
LIN {X 0,Y 601.417,Z 152.568,A -85,B 0,C 180,E1 -556.987,E2 -556.987} C_VEL
LIN {X 0,Y 601.4,Z 152.57,A -85,B 0,C 180,E1 -559.81,E2 -559.81} C_VEL
LIN {X 0,Y 601.409,Z 152.574,A -85,B 0,C 180,E1 -562.683,E2 -562.683} C_VEL
LIN {X 0,Y 601.371,Z 152.573,A -85,B 0,C 180,E1 -564.88,E2 -564.88} C_VEL
LIN {X 0,Y 601.408,Z 152.572,A -85,B 0,C 180,E1 -567.868,E2 -567.868} C_VEL
LIN {X 0,Y 601.427,Z 152.566,A -85,B 0,C 180,E1 -570.164,E2 -570.164} C_VEL
LIN {X 0,Y 601.414,Z 152.574,A -85,B 0,C 180,E1 -572.72,E2 -572.72} C_VEL
LIN {X 0,Y 601.375,Z 152.572,A -85,B 0,C 180,E1 -575.114,E2 -575.114} C_VEL
LIN {X 0,Y 601.41,Z 152.571,A -85,B 0,C 180,E1 -577.421,E2 -577.421} C_VEL
LIN {X 0,Y 601.394,Z 152.57,A -85,B 0,C 180,E1 -579.997,E2 -579.997} C_VEL
LIN {X 0,Y 601.401,Z 152.575,A -85,B 0,C 180,E1 -582.672,E2 -582.672} C_VEL
LIN {X 0,Y 601.412,Z 152.568,A -85,B 0,C 180,E1 -585.484,E2 -585.484} C_VEL
LIN {X 0,Y 601.402,Z 152.569,A -85,B 0,C 180,E1 -588.41,E2 -588.41} C_VEL
LIN {X 0,Y 601.387,Z 152.574,A -85,B 0,C 180,E1 -590.874,E2 -590.874} C_VEL
LIN {X 0,Y 601.397,Z 152.574,A -85,B 0,C 180,E1 -592.624,E2 -592.624} C_VEL
LIN {X 0,Y 601.412,Z 156.679,A -85,B 0,C 180,E1 -595.07,E2 -595.07} C_VEL
LIN {X 0,Y 601.396,Z 160.901,A -85,B 0,C 180,E1 -597.484,E2 -597.484} C_VEL
LIN {X 0,Y 601.379,Z 166.451,A -85,B 0,C 180,E1 -600.607,E2 -600.607} C_VEL
LIN {X 0,Y 601.383,Z 170.601,A -85,B 0,C 180,E1 -602.887,E2 -602.887} C_VEL
LIN {X 0,Y 601.374,Z 176.219,A -85,B 0,C 180,E1 -605.857,E2 -605.857} C_VEL
LIN {X 0,Y 601.336,Z 180.424,A -85,B 0,C 180,E1 -608.039,E2 -608.039} C_VEL
LIN {X 0,Y 601.326,Z 184.624,A -85,B 0,C 180,E1 -610.189,E2 -610.189} C_VEL
LIN {X 0,Y 601.333,Z 190.214,A -85,B 0,C 180,E1 -613.012,E2 -613.012} C_VEL
LIN {X 0,Y 601.32,Z 196.11,A -85,B 0,C 180,E1 -615.949,E2 -615.949} C_VEL
LIN {X 0,Y 601.317,Z 196.527,A -85,B 0,C 180,E1 -616.156,E2 -616.156} C_VEL
LIN {X 0,Y 601.594,Z 200.837,A -85,B 0,C 180,E1 -616.257,E2 -616.257} C_VEL
LIN {X 0,Y 601.575,Z 213.409,A -85,B 0,C 180,E1 -616.574,E2 -616.574} C_VEL
LIN {X 0,Y 601.502,Z 225.225,A -85,B 0,C 180,E1 -617.002,E2 -617.002} C_VEL
LIN {X 0,Y 601.443,Z 237.622,A -85,B 0,C 180,E1 -617.602,E2 -617.602} C_VEL
LIN {X 0,Y 601.481,Z 248.693,A -85,B 0,C 180,E1 -618.287,E2 -618.287} C_VEL
LIN {X 0,Y 601.436,Z 259.489,A -85,B 0,C 180,E1 -619.128,E2 -619.128} C_VEL
LIN {X 0,Y 601.408,Z 269.286,A -85,B 0,C 180,E1 -620.075,E2 -620.075} C_VEL
LIN {X 0,Y 601.389,Z 277.701,A -85,B 0,C 180,E1 -621.092,E2 -621.092} C_VEL
LIN {X 0,Y 601.361,Z 284.467,A -85,B 0,C 180,E1 -622.107,E2 -622.107} C_VEL
LIN {X 0,Y 601.361,Z 290.668,A -85,B 0,C 180,E1 -623.289,E2 -623.289} C_VEL
LIN {X 0,Y 601.357,Z 294.687,A -85,B 0,C 180,E1 -624.299,E2 -624.299} C_VEL
LIN {X 0,Y 601.329,Z 297.658,A -85,B 0,C 180,E1 -625.307,E2 -625.307} C_VEL
LIN {X 0,Y 601.343,Z 299.107,A -85,B 0,C 180,E1 -625.979,E2 -625.979} C_VEL
LIN {X 0,Y 601.32,Z 300.745,A -85,B 0,C 180,E1 -627.32,E2 -627.32} C_VEL
LIN {X 0,Y 601.343,Z 300.993,A -85,B 0,C 180,E1 -627.99,E2 -627.99} C_VEL
LIN {X 0,Y 601.347,Z 300.822,A -85,B 0,C 180,E1 -628.66,E2 -628.66} C_VEL
LIN {X 0,Y 601.338,Z 299.292,A -85,B 0,C 180,E1 -630,E2 -630} C_VEL
LIN {X 0,Y 601.338,Z 297.94,A -85,B 0,C 180,E1 -630.669,E2 -630.669} C_VEL
LIN {X 0,Y 601.358,Z 295.077,A -85,B 0,C 180,E1 -631.674,E2 -631.674} C_VEL
LIN {X 0,Y 601.337,Z 291.199,A -85,B 0,C 180,E1 -632.679,E2 -632.679} C_VEL
LIN {X 0,Y 601.368,Z 286.198,A -85,B 0,C 180,E1 -633.685,E2 -633.685} C_VEL
LIN {X 0,Y 601.401,Z 279.926,A -85,B 0,C 180,E1 -634.691,E2 -634.691} C_VEL
LIN {X 0,Y 601.399,Z 272.081,A -85,B 0,C 180,E1 -635.7,E2 -635.7} C_VEL
LIN {X 0,Y 601.437,Z 262.325,A -85,B 0,C 180,E1 -636.71,E2 -636.71} C_VEL
LIN {X 0,Y 601.457,Z 252.15,A -85,B 0,C 180,E1 -637.553,E2 -637.553} C_VEL
LIN {X 0,Y 601.459,Z 240.7,A -85,B 0,C 180,E1 -638.313,E2 -638.313} C_VEL
LIN {X 0,Y 601.485,Z 229.413,A -85,B 0,C 180,E1 -638.905,E2 -638.905} C_VEL
LIN {X 0,Y 601.537,Z 217.845,A -85,B 0,C 180,E1 -639.37,E2 -639.37} C_VEL
LIN {X 0,Y 601.605,Z 204.561,A -85,B 0,C 180,E1 -639.751,E2 -639.751} C_VEL
LIN {X 0,Y 601.34,Z 196.544,A -85,B 0,C 180,E1 -639.925,E2 -639.925} C_VEL
LIN {X 0,Y 601.304,Z 190.712,A -85,B 0,C 180,E1 -642.829,E2 -642.829} C_VEL
LIN {X 0,Y 601.326,Z 185.232,A -85,B 0,C 180,E1 -645.592,E2 -645.592} C_VEL
LIN {X 0,Y 601.349,Z 179.762,A -85,B 0,C 180,E1 -648.392,E2 -648.392} C_VEL
LIN {X 0,Y 601.36,Z 174.302,A -85,B 0,C 180,E1 -651.239,E2 -651.239} C_VEL
LIN {X 0,Y 601.382,Z 168.854,A -85,B 0,C 180,E1 -654.141,E2 -654.141} C_VEL
LIN {X 0,Y 601.358,Z 164.87,A -85,B 0,C 180,E1 -656.363,E2 -656.363} C_VEL
LIN {X 0,Y 601.376,Z 160.605,A -85,B 0,C 180,E1 -658.777,E2 -658.777} C_VEL
LIN {X 0,Y 601.389,Z 155.929,A -85,B 0,C 180,E1 -661.449,E2 -661.449} C_VEL
LIN {X 0,Y 601.355,Z 152.751,A -85,B 0,C 180,E1 -663.315,E2 -663.315} C_VEL
LIN {X 0,Y 601.386,Z 152.577,A -85,B 0,C 180,E1 -665.11,E2 -665.11} C_VEL
LIN {X 0,Y 601.414,Z 152.567,A -85,B 0,C 180,E1 -667.417,E2 -667.417} C_VEL
LIN {X 0,Y 601.392,Z 152.574,A -85,B 0,C 180,E1 -669.993,E2 -669.993} C_VEL
LIN {X 0,Y 601.423,Z 152.566,A -85,B 0,C 180,E1 -672.665,E2 -672.665} C_VEL
LIN {X 0,Y 601.405,Z 152.576,A -85,B 0,C 180,E1 -675.479,E2 -675.479} C_VEL
LIN {X 0,Y 601.416,Z 152.567,A -85,B 0,C 180,E1 -678.402,E2 -678.402} C_VEL
LIN {X 0,Y 601.415,Z 152.572,A -85,B 0,C 180,E1 -680.873,E2 -680.873} C_VEL
LIN {X 0,Y 601.389,Z 152.572,A -85,B 0,C 180,E1 -683.735,E2 -683.735} C_VEL
LIN {X 0,Y 601.407,Z 152.568,A -85,B 0,C 180,E1 -686.685,E2 -686.685} C_VEL
LIN {X 0,Y 601.41,Z 152.57,A -85,B 0,C 180,E1 -689.057,E2 -689.057} C_VEL
LIN {X 0,Y 601.427,Z 152.57,A -85,B 0,C 180,E1 -691.373,E2 -691.373} C_VEL
LIN {X 0,Y 601.398,Z 152.569,A -85,B 0,C 180,E1 -693.636,E2 -693.636} C_VEL
LIN {X 0,Y 601.407,Z 152.572,A -85,B 0,C 180,E1 -696.589,E2 -696.589} C_VEL
LIN {X 0,Y 601.411,Z 152.57,A -85,B 0,C 180,E1 -699.477,E2 -699.477} C_VEL
LIN {X 0,Y 601.356,Z 152.574,A -85,B 0,C 180,E1 -702.31,E2 -702.31} C_VEL
LIN {X 0,Y 601.388,Z 152.57,A -85,B 0,C 180,E1 -704.408,E2 -704.408} C_VEL
LIN {X 0,Y 601.445,Z 152.566,A -85,B 0,C 180,E1 -707.172,E2 -707.172} C_VEL
LIN {X 0,Y 601.429,Z 152.567,A -85,B 0,C 180,E1 -709.905,E2 -709.905} C_VEL
LIN {X 0,Y 601.427,Z 152.566,A -85,B 0,C 180,E1 -712.615,E2 -712.615} C_VEL
LIN {X 0,Y 601.422,Z 152.57,A -85,B 0,C 180,E1 -715.308,E2 -715.308} C_VEL
LIN {X 0,Y 601.375,Z 152.572,A -85,B 0,C 180,E1 -717.991,E2 -717.991} C_VEL
LIN {X 0,Y 601.438,Z 152.57,A -85,B 0,C 180,E1 -720.669,E2 -720.669} C_VEL
LIN {X 0,Y 601.409,Z 152.567,A -85,B 0,C 180,E1 -723.35,E2 -723.35} C_VEL
LIN {X 0,Y 601.432,Z 152.573,A -85,B 0,C 180,E1 -726.037,E2 -726.037} C_VEL
LIN {X 0,Y 601.429,Z 152.565,A -85,B 0,C 180,E1 -728.738,E2 -728.738} C_VEL
LIN {X 0,Y 601.413,Z 152.572,A -85,B 0,C 180,E1 -731.458,E2 -731.458} C_VEL
LIN {X 0,Y 601.391,Z 152.571,A -85,B 0,C 180,E1 -733.516,E2 -733.516} C_VEL
LIN {X 0,Y 601.413,Z 152.572,A -85,B 0,C 180,E1 -736.288,E2 -736.288} C_VEL
LIN {X 0,Y 601.385,Z 152.57,A -85,B 0,C 180,E1 -739.1,E2 -739.1} C_VEL
LIN {X 0,Y 601.385,Z 152.572,A -85,B 0,C 180,E1 -741.24,E2 -741.24} C_VEL
LIN {X 0,Y 601.453,Z 152.562,A -85,B 0,C 180,E1 -744.141,E2 -744.141} C_VEL
LIN {X 0,Y 601.44,Z 152.569,A -85,B 0,C 180,E1 -747.112,E2 -747.112} C_VEL
LIN {X 0,Y 601.406,Z 152.568,A -85,B 0,C 180,E1 -749.394,E2 -749.394} C_VEL
LIN {X 0,Y 601.391,Z 152.572,A -85,B 0,C 180,E1 -751.728,E2 -751.728} C_VEL
LIN {X 0,Y 601.397,Z 152.574,A -85,B 0,C 180,E1 -754.12,E2 -754.12} C_VEL
LIN {X 0,Y 601.381,Z 152.571,A -85,B 0,C 180,E1 -756.585,E2 -756.585} C_VEL
LIN {X 0,Y 601.431,Z 152.567,A -85,B 0,C 180,E1 -759.54,E2 -759.54} C_VEL
LIN {X 0,Y 601.42,Z 152.574,A -85,B 0,C 180,E1 -762.597,E2 -762.597} C_VEL
LIN {X 0,Y 601.403,Z 152.568,A -85,B 0,C 180,E1 -765.485,E2 -765.485} C_VEL
LIN {X 0,Y 601.404,Z 152.57,A -85,B 0,C 180,E1 -768.409,E2 -768.409} C_VEL
LIN {X 0,Y 601.378,Z 152.573,A -85,B 0,C 180,E1 -770.875,E2 -770.875} C_VEL
LIN {X 0,Y 601.389,Z 152.575,A -85,B 0,C 180,E1 -773.42,E2 -773.42} C_VEL
LIN {X 0,Y 601.406,Z 152.666,A -85,B 0,C 180,E1 -774.336,E2 -774.336} C_VEL
LIN {X 0,Y 601.523,Z 159.066,A -85,B 0,C 180,E1 -776.696,E2 -776.696} C_VEL
LIN {X 0,Y 601.471,Z 166.844,A -85,B 0,C 180,E1 -779.453,E2 -779.453} C_VEL
LIN {X 0,Y 601.435,Z 174.73,A -85,B 0,C 180,E1 -782.136,E2 -782.136} C_VEL
LIN {X 0,Y 601.438,Z 182.551,A -85,B 0,C 180,E1 -784.756,E2 -784.756} C_VEL
LIN {X 0,Y 601.412,Z 190.577,A -85,B 0,C 180,E1 -787.396,E2 -787.396} C_VEL
LIN {X 0,Y 601.391,Z 199.245,A -85,B 0,C 180,E1 -790.192,E2 -790.192} C_VEL
LIN {X 0,Y 601.372,Z 208.149,A -85,B 0,C 180,E1 -793.014,E2 -793.014} C_VEL
LIN {X 0,Y 601.364,Z 217.493,A -85,B 0,C 180,E1 -795.931,E2 -795.931} C_VEL
LIN {X 0,Y 601.362,Z 224.496,A -85,B 0,C 180,E1 -798.093,E2 -798.093} C_VEL
LIN {X 0,Y 601.612,Z 232.581,A -85,B 0,C 180,E1 -798.248,E2 -798.248} C_VEL
LIN {X 0,Y 601.55,Z 245.048,A -85,B 0,C 180,E1 -798.583,E2 -798.583} C_VEL
LIN {X 0,Y 601.493,Z 257.467,A -85,B 0,C 180,E1 -799.054,E2 -799.054} C_VEL
LIN {X 0,Y 601.441,Z 269.348,A -85,B 0,C 180,E1 -799.651,E2 -799.651} C_VEL
LIN {X 0,Y 601.46,Z 279.948,A -85,B 0,C 180,E1 -800.331,E2 -800.331} C_VEL
LIN {X 0,Y 601.434,Z 289.612,A -85,B 0,C 180,E1 -801.094,E2 -801.094} C_VEL
LIN {X 0,Y 601.406,Z 298.423,A -85,B 0,C 180,E1 -801.94,E2 -801.94} C_VEL
LIN {X 0,Y 601.383,Z 307.006,A -85,B 0,C 180,E1 -802.953,E2 -802.953} C_VEL
LIN {X 0,Y 601.36,Z 313.872,A -85,B 0,C 180,E1 -803.963,E2 -803.963} C_VEL
LIN {X 0,Y 601.345,Z 319.369,A -85,B 0,C 180,E1 -804.972,E2 -804.972} C_VEL
LIN {X 0,Y 601.346,Z 323.679,A -85,B 0,C 180,E1 -805.98,E2 -805.98} C_VEL
LIN {X 0,Y 601.344,Z 325.958,A -85,B 0,C 180,E1 -806.651,E2 -806.651} C_VEL
LIN {X 0,Y 601.325,Z 327.811,A -85,B 0,C 180,E1 -807.321,E2 -807.321} C_VEL
LIN {X 0,Y 601.343,Z 329.203,A -85,B 0,C 180,E1 -807.991,E2 -807.991} C_VEL
LIN {X 0,Y 601.339,Z 330.784,A -85,B 0,C 180,E1 -809.331,E2 -809.331} C_VEL
LIN {X 0,Y 601.335,Z 331,A -85,B 0,C 180,E1 -810,E2 -810} C_VEL
LIN {X 0,Y 601.347,Z 330.184,A -85,B 0,C 180,E1 -811.34,E2 -811.34} C_VEL
LIN {X 0,Y 601.343,Z 329.201,A -85,B 0,C 180,E1 -812.01,E2 -812.01} C_VEL
LIN {X 0,Y 601.325,Z 327.809,A -85,B 0,C 180,E1 -812.68,E2 -812.68} C_VEL
LIN {X 0,Y 601.368,Z 324.895,A -85,B 0,C 180,E1 -813.686,E2 -813.686} C_VEL
LIN {X 0,Y 601.336,Z 320.949,A -85,B 0,C 180,E1 -814.693,E2 -814.693} C_VEL
LIN {X 0,Y 601.372,Z 314.877,A -85,B 0,C 180,E1 -815.869,E2 -815.869} C_VEL
LIN {X 0,Y 601.382,Z 308.236,A -85,B 0,C 180,E1 -816.88,E2 -816.88} C_VEL
LIN {X 0,Y 601.4,Z 299.99,A -85,B 0,C 180,E1 -817.892,E2 -817.892} C_VEL
LIN {X 0,Y 601.436,Z 291.539,A -85,B 0,C 180,E1 -818.737,E2 -818.737} C_VEL
LIN {X 0,Y 601.446,Z 281.096,A -85,B 0,C 180,E1 -819.585,E2 -819.585} C_VEL
LIN {X 0,Y 601.441,Z 270.762,A -85,B 0,C 180,E1 -820.265,E2 -820.265} C_VEL
LIN {X 0,Y 601.477,Z 259.296,A -85,B 0,C 180,E1 -820.866,E2 -820.866} C_VEL
LIN {X 0,Y 601.523,Z 246.358,A -85,B 0,C 180,E1 -821.375,E2 -821.375} C_VEL
LIN {X 0,Y 601.604,Z 233.455,A -85,B 0,C 180,E1 -821.732,E2 -821.732} C_VEL
LIN {X 0,Y 601.493,Z 225.642,A -85,B 0,C 180,E1 -821.884,E2 -821.884} C_VEL
LIN {X 0,Y 601.333,Z 224.423,A -85,B 0,C 180,E1 -821.93,E2 -821.93} C_VEL
LIN {X 0,Y 601.336,Z 215.937,A -85,B 0,C 180,E1 -824.552,E2 -824.552} C_VEL
LIN {X 0,Y 601.392,Z 207.033,A -85,B 0,C 180,E1 -827.337,E2 -827.337} C_VEL
LIN {X 0,Y 601.371,Z 198.129,A -85,B 0,C 180,E1 -830.166,E2 -830.166} C_VEL
LIN {X 0,Y 601.429,Z 189.226,A -85,B 0,C 180,E1 -833.044,E2 -833.044} C_VEL
LIN {X 0,Y 601.413,Z 180.686,A -85,B 0,C 180,E1 -835.867,E2 -835.867} C_VEL
LIN {X 0,Y 601.449,Z 172.457,A -85,B 0,C 180,E1 -838.624,E2 -838.624} C_VEL
LIN {X 0,Y 601.483,Z 164.212,A -85,B 0,C 180,E1 -841.464,E2 -841.464} C_VEL
LIN {X 0,Y 601.466,Z 156.84,A -85,B 0,C 180,E1 -844.114,E2 -844.114} C_VEL
LIN {X 0,Y 601.404,Z 152.573,A -85,B 0,C 180,E1 -845.708,E2 -845.708} C_VEL
LIN {X 0,Y 601.394,Z 152.577,A -85,B 0,C 180,E1 -848.466,E2 -848.466} C_VEL
LIN {X 0,Y 601.408,Z 152.568,A -85,B 0,C 180,E1 -850.872,E2 -850.872} C_VEL
LIN {X 0,Y 601.435,Z 152.572,A -85,B 0,C 180,E1 -853.582,E2 -853.582} C_VEL
LIN {X 0,Y 601.434,Z 152.566,A -85,B 0,C 180,E1 -856.423,E2 -856.423} C_VEL
LIN {X 0,Y 601.384,Z 152.571,A -85,B 0,C 180,E1 -859.426,E2 -859.426} C_VEL
LIN {X 0,Y 601.404,Z 152.573,A -85,B 0,C 180,E1 -861.731,E2 -861.731} C_VEL
LIN {X 0,Y 601.397,Z 152.57,A -85,B 0,C 180,E1 -864.246,E2 -864.246} C_VEL
LIN {X 0,Y 601.419,Z 152.569,A -85,B 0,C 180,E1 -866.686,E2 -866.686} C_VEL
LIN {X 0,Y 601.414,Z 152.57,A -85,B 0,C 180,E1 -869.058,E2 -869.058} C_VEL
LIN {X 0,Y 601.401,Z 152.569,A -85,B 0,C 180,E1 -871.372,E2 -871.372} C_VEL
LIN {X 0,Y 601.384,Z 152.574,A -85,B 0,C 180,E1 -874.131,E2 -874.131} C_VEL
LIN {X 0,Y 601.406,Z 152.569,A -85,B 0,C 180,E1 -876.589,E2 -876.589} C_VEL
LIN {X 0,Y 601.424,Z 152.566,A -85,B 0,C 180,E1 -879.478,E2 -879.478} C_VEL
LIN {X 0,Y 601.386,Z 152.576,A -85,B 0,C 180,E1 -882.311,E2 -882.311} C_VEL
LIN {X 0,Y 601.39,Z 152.571,A -85,B 0,C 180,E1 -884.408,E2 -884.408} C_VEL
LIN {X 0,Y 601.404,Z 152.576,A -85,B 0,C 180,E1 -887.172,E2 -887.172} C_VEL
LIN {X 0,Y 601.426,Z 152.569,A -85,B 0,C 180,E1 -889.224,E2 -889.224} C_VEL
LIN {X 0,Y 601.431,Z 152.568,A -85,B 0,C 180,E1 -891.939,E2 -891.939} C_VEL
LIN {X 0,Y 601.431,Z 152.573,A -85,B 0,C 180,E1 -893.963,E2 -893.963} C_VEL
LIN {X 0,Y 601.402,Z 152.569,A -85,B 0,C 180,E1 -896.65,E2 -896.65} C_VEL
LIN {X 0,Y 601.425,Z 152.569,A -85,B 0,C 180,E1 -899.331,E2 -899.331} C_VEL
LIN {X 0,Y 601.404,Z 152.571,A -85,B 0,C 180,E1 -902.009,E2 -902.009} C_VEL
LIN {X 0,Y 601.421,Z 152.567,A -85,B 0,C 180,E1 -904.692,E2 -904.692} C_VEL
LIN {X 0,Y 601.436,Z 152.572,A -85,B 0,C 180,E1 -907.385,E2 -907.385} C_VEL
LIN {X 0,Y 601.403,Z 152.569,A -85,B 0,C 180,E1 -910.096,E2 -910.096} C_VEL
LIN {X 0,Y 601.384,Z 152.573,A -85,B 0,C 180,E1 -912.403,E2 -912.403} C_VEL
LIN {X 0,Y 600.729,Z 152.655,A -85,B 0,C 180,E1 -912.963,E2 -912.963} C_VEL
LIN {X 0,Y 597.88,Z 153.011,A -85,B 0,C 180,E1 -913.871,E2 -913.871} C_VEL
LIN {X 0,Y 595.468,Z 153.31,A -85,B 0,C 180,E1 -914.601,E2 -914.601} C_VEL
LIN {X 0,Y 594.434,Z 153.437,A -85,B 0,C 180,E1 -915.165,E2 -915.165} C_VEL
LIN {X 0,Y 594.351,Z 153.449,A -85,B 0,C 180,E1 -915.356,E2 -915.356} C_VEL
LIN {X 0,Y 594.37,Z 153.447,A -85,B 0,C 180,E1 -917.905,E2 -917.905} C_VEL
LIN {X 0,Y 594.37,Z 153.452,A -85,B 0,C 180,E1 -920.923,E2 -920.923} C_VEL
LIN {X 0,Y 594.368,Z 153.446,A -85,B 0,C 180,E1 -923.705,E2 -923.705} C_VEL
LIN {X 0,Y 594.36,Z 153.446,A -85,B 0,C 180,E1 -926.701,E2 -926.701} C_VEL
LIN {X 0,Y 594.366,Z 153.449,A -85,B 0,C 180,E1 -929,E2 -929} C_VEL
LIN {X 0,Y 594.378,Z 153.444,A -85,B 0,C 180,E1 -931.649,E2 -931.649} C_VEL
LIN {X 0,Y 594.36,Z 153.45,A -85,B 0,C 180,E1 -934.582,E2 -934.582} C_VEL
LIN {X 0,Y 594.365,Z 153.452,A -85,B 0,C 180,E1 -937.61,E2 -937.61} C_VEL
LIN {X 0,Y 594.354,Z 153.448,A -85,B 0,C 180,E1 -940.569,E2 -940.569} C_VEL
LIN {X 0,Y 594.366,Z 153.446,A -85,B 0,C 180,E1 -943.3,E2 -943.3} C_VEL
LIN {X 0,Y 594.355,Z 153.454,A -85,B 0,C 180,E1 -946.162,E2 -946.162} C_VEL
LIN {X 0,Y 594.36,Z 153.446,A -85,B 0,C 180,E1 -948.537,E2 -948.537} C_VEL
LIN {X 0,Y 594.36,Z 153.452,A -85,B 0,C 180,E1 -951.299,E2 -951.299} C_VEL
LIN {X 0,Y 594.354,Z 153.449,A -85,B 0,C 180,E1 -952.397,E2 -952.397} C_VEL
LIN {X 0,Y 594.329,Z 153.841,A -85,B 0,C 180,E1 -952.912,E2 -952.912} C_VEL
LIN {X 0,Y 594.32,Z 158.873,A -85,B 0,C 180,E1 -955.871,E2 -955.871} C_VEL
LIN {X 0,Y 594.322,Z 163.691,A -85,B 0,C 180,E1 -958.649,E2 -958.649} C_VEL
LIN {X 0,Y 594.293,Z 167.962,A -85,B 0,C 180,E1 -961.059,E2 -961.059} C_VEL
LIN {X 0,Y 594.285,Z 171.953,A -85,B 0,C 180,E1 -963.297,E2 -963.297} C_VEL
LIN {X 0,Y 594.305,Z 176.23,A -85,B 0,C 180,E1 -965.585,E2 -965.585} C_VEL
LIN {X 0,Y 594.264,Z 180.373,A -85,B 0,C 180,E1 -967.764,E2 -967.764} C_VEL
LIN {X 0,Y 594.234,Z 184.573,A -85,B 0,C 180,E1 -969.942,E2 -969.942} C_VEL
LIN {X 0,Y 594.224,Z 188.767,A -85,B 0,C 180,E1 -972.092,E2 -972.092} C_VEL
LIN {X 0,Y 594.21,Z 194.35,A -85,B 0,C 180,E1 -974.918,E2 -974.918} C_VEL
LIN {X 0,Y 594.222,Z 196.751,A -85,B 0,C 180,E1 -976.031,E2 -976.031} C_VEL
LIN {X 0,Y 594.66,Z 201.898,A -85,B 0,C 180,E1 -976.138,E2 -976.138} C_VEL
LIN {X 0,Y 594.623,Z 213.998,A -85,B 0,C 180,E1 -976.458,E2 -976.458} C_VEL
LIN {X 0,Y 594.522,Z 226.662,A -85,B 0,C 180,E1 -976.934,E2 -976.934} C_VEL
LIN {X 0,Y 594.456,Z 238.766,A -85,B 0,C 180,E1 -977.54,E2 -977.54} C_VEL
LIN {X 0,Y 594.458,Z 249.559,A -85,B 0,C 180,E1 -978.233,E2 -978.233} C_VEL
LIN {X 0,Y 594.391,Z 260.321,A -85,B 0,C 180,E1 -979.095,E2 -979.095} C_VEL
LIN {X 0,Y 594.35,Z 269.062,A -85,B 0,C 180,E1 -979.956,E2 -979.956} C_VEL
LIN {X 0,Y 594.313,Z 277.53,A -85,B 0,C 180,E1 -980.986,E2 -980.986} C_VEL
LIN {X 0,Y 594.295,Z 284.327,A -85,B 0,C 180,E1 -982.013,E2 -982.013} C_VEL
LIN {X 0,Y 594.281,Z 290.559,A -85,B 0,C 180,E1 -983.208,E2 -983.208} C_VEL
LIN {X 0,Y 594.267,Z 294.603,A -85,B 0,C 180,E1 -984.231,E2 -984.231} C_VEL
LIN {X 0,Y 594.229,Z 297.597,A -85,B 0,C 180,E1 -985.251,E2 -985.251} C_VEL
LIN {X 0,Y 594.256,Z 299.067,A -85,B 0,C 180,E1 -985.931,E2 -985.931} C_VEL
LIN {X 0,Y 594.259,Z 300.093,A -85,B 0,C 180,E1 -986.61,E2 -986.61} C_VEL
LIN {X 0,Y 594.241,Z 300.988,A -85,B 0,C 180,E1 -987.966,E2 -987.966} C_VEL
LIN {X 0,Y 594.247,Z 300.838,A -85,B 0,C 180,E1 -988.644,E2 -988.644} C_VEL
LIN {X 0,Y 594.238,Z 299.33,A -85,B 0,C 180,E1 -990,E2 -990} C_VEL
LIN {X 0,Y 594.239,Z 297.989,A -85,B 0,C 180,E1 -990.677,E2 -990.677} C_VEL
LIN {X 0,Y 594.28,Z 295.15,A -85,B 0,C 180,E1 -991.694,E2 -991.694} C_VEL
LIN {X 0,Y 594.243,Z 291.297,A -85,B 0,C 180,E1 -992.711,E2 -992.711} C_VEL
LIN {X 0,Y 594.29,Z 286.323,A -85,B 0,C 180,E1 -993.729,E2 -993.729} C_VEL
LIN {X 0,Y 594.339,Z 280.082,A -85,B 0,C 180,E1 -994.747,E2 -994.747} C_VEL
LIN {X 0,Y 594.33,Z 272.286,A -85,B 0,C 180,E1 -995.768,E2 -995.768} C_VEL
LIN {X 0,Y 594.393,Z 262.57,A -85,B 0,C 180,E1 -996.789,E2 -996.789} C_VEL
LIN {X 0,Y 594.436,Z 252.471,A -85,B 0,C 180,E1 -997.642,E2 -997.642} C_VEL
LIN {X 0,Y 594.446,Z 241.09,A -85,B 0,C 180,E1 -998.412,E2 -998.412} C_VEL
LIN {X 0,Y 594.503,Z 229.898,A -85,B 0,C 180,E1 -999.011,E2 -999.011} C_VEL
LIN {X 0,Y 594.583,Z 218.533,A -85,B 0,C 180,E1 -999.481,E2 -999.481} C_VEL
LIN {X 0,Y 594.662,Z 205.562,A -85,B 0,C 180,E1 -999.866,E2 -999.866} C_VEL
LIN {X 0,Y 594.531,Z 198.53,A -85,B 0,C 180,E1 -1000.019,E2 -1000.019} C_VEL
LIN {X 0,Y 594.228,Z 196.507,A -85,B 0,C 180,E1 -1000.088,E2 -1000.088} C_VEL
LIN {X 0,Y 594.226,Z 190.76,A -85,B 0,C 180,E1 -1002.985,E2 -1002.985} C_VEL
LIN {X 0,Y 594.252,Z 185.281,A -85,B 0,C 180,E1 -1005.782,E2 -1005.782} C_VEL
LIN {X 0,Y 594.263,Z 181.178,A -85,B 0,C 180,E1 -1007.906,E2 -1007.906} C_VEL
LIN {X 0,Y 594.249,Z 177.082,A -85,B 0,C 180,E1 -1010.056,E2 -1010.056} C_VEL
LIN {X 0,Y 594.309,Z 172.084,A -85,B 0,C 180,E1 -1012.721,E2 -1012.721} C_VEL
LIN {X 0,Y 594.311,Z 167.661,A -85,B 0,C 180,E1 -1015.194,E2 -1015.194} C_VEL
LIN {X 0,Y 594.335,Z 163.576,A -85,B 0,C 180,E1 -1017.516,E2 -1017.516} C_VEL
LIN {X 0,Y 594.337,Z 158.69,A -85,B 0,C 180,E1 -1020.319,E2 -1020.319} C_VEL
LIN {X 0,Y 594.328,Z 154.218,A -85,B 0,C 180,E1 -1022.95,E2 -1022.95} C_VEL
LIN {X 0,Y 594.333,Z 153.451,A -85,B 0,C 180,E1 -1023.761,E2 -1023.761} C_VEL
LIN {X 0,Y 594.35,Z 153.451,A -85,B 0,C 180,E1 -1026.478,E2 -1026.478} C_VEL
LIN {X 0,Y 594.36,Z 153.449,A -85,B 0,C 180,E1 -1028.803,E2 -1028.803} C_VEL
LIN {X 0,Y 594.367,Z 153.446,A -85,B 0,C 180,E1 -1031.461,E2 -1031.461} C_VEL
LIN {X 0,Y 594.362,Z 153.447,A -85,B 0,C 180,E1 -1034.233,E2 -1034.233} C_VEL
LIN {X 0,Y 594.365,Z 153.452,A -85,B 0,C 180,E1 -1037.143,E2 -1037.143} C_VEL
LIN {X 0,Y 594.353,Z 153.448,A -85,B 0,C 180,E1 -1039.431,E2 -1039.431} C_VEL
LIN {X 0,Y 594.362,Z 153.453,A -85,B 0,C 180,E1 -1042.389,E2 -1042.389} C_VEL
LIN {X 0,Y 594.345,Z 153.449,A -85,B 0,C 180,E1 -1045.417,E2 -1045.417} C_VEL
LIN {X 0,Y 594.371,Z 153.445,A -85,B 0,C 180,E1 -1048.351,E2 -1048.351} C_VEL
LIN {X 0,Y 594.394,Z 153.448,A -85,B 0,C 180,E1 -1051.032,E2 -1051.032} C_VEL
LIN {X 0,Y 594.368,Z 153.445,A -85,B 0,C 180,E1 -1054.055,E2 -1054.055} C_VEL
LIN {X 0,Y 594.379,Z 153.45,A -85,B 0,C 180,E1 -1056.295,E2 -1056.295} C_VEL
LIN {X 0,Y 594.376,Z 153.444,A -85,B 0,C 180,E1 -1059.223,E2 -1059.223} C_VEL
LIN {X 0,Y 594.316,Z 153.453,A -85,B 0,C 180,E1 -1062.094,E2 -1062.094} C_VEL
LIN {X 0,Y 594.346,Z 153.447,A -85,B 0,C 180,E1 -1064.218,E2 -1064.218} C_VEL
LIN {X 0,Y 594.383,Z 153.448,A -85,B 0,C 180,E1 -1067.017,E2 -1067.017} C_VEL
LIN {X 0,Y 594.388,Z 153.443,A -85,B 0,C 180,E1 -1069.784,E2 -1069.784} C_VEL
LIN {X 0,Y 594.389,Z 153.444,A -85,B 0,C 180,E1 -1072.527,E2 -1072.527} C_VEL
LIN {X 0,Y 594.388,Z 153.445,A -85,B 0,C 180,E1 -1075.252,E2 -1075.252} C_VEL
LIN {X 0,Y 594.347,Z 153.448,A -85,B 0,C 180,E1 -1077.967,E2 -1077.967} C_VEL
LIN {X 0,Y 594.405,Z 153.446,A -85,B 0,C 180,E1 -1080.677,E2 -1080.677} C_VEL
LIN {X 0,Y 594.36,Z 153.446,A -85,B 0,C 180,E1 -1083.389,E2 -1083.389} C_VEL
LIN {X 0,Y 594.385,Z 153.449,A -85,B 0,C 180,E1 -1086.109,E2 -1086.109} C_VEL
LIN {X 0,Y 594.387,Z 153.442,A -85,B 0,C 180,E1 -1088.842,E2 -1088.842} C_VEL
LIN {X 0,Y 594.367,Z 153.448,A -85,B 0,C 180,E1 -1091.596,E2 -1091.596} C_VEL
LIN {X 0,Y 594.359,Z 153.449,A -85,B 0,C 180,E1 -1094.378,E2 -1094.378} C_VEL
LIN {X 0,Y 594.351,Z 153.447,A -85,B 0,C 180,E1 -1097.194,E2 -1097.194} C_VEL
LIN {X 0,Y 594.354,Z 153.453,A -85,B 0,C 180,E1 -1100.054,E2 -1100.054} C_VEL
LIN {X 0,Y 594.387,Z 153.444,A -85,B 0,C 180,E1 -1102.966,E2 -1102.966} C_VEL
LIN {X 0,Y 594.364,Z 153.453,A -85,B 0,C 180,E1 -1105.194,E2 -1105.194} C_VEL
LIN {X 0,Y 594.358,Z 153.446,A -85,B 0,C 180,E1 -1107.53,E2 -1107.53} C_VEL
LIN {X 0,Y 594.367,Z 153.445,A -85,B 0,C 180,E1 -1109.777,E2 -1109.777} C_VEL
LIN {X 0,Y 594.345,Z 153.455,A -85,B 0,C 180,E1 -1112.148,E2 -1112.148} C_VEL
LIN {X 0,Y 594.343,Z 153.448,A -85,B 0,C 180,E1 -1114.582,E2 -1114.582} C_VEL
LIN {X 0,Y 594.358,Z 153.449,A -85,B 0,C 180,E1 -1117.089,E2 -1117.089} C_VEL
LIN {X 0,Y 594.363,Z 153.446,A -85,B 0,C 180,E1 -1119.779,E2 -1119.779} C_VEL
LIN {X 0,Y 594.369,Z 153.448,A -85,B 0,C 180,E1 -1122.375,E2 -1122.375} C_VEL
LIN {X 0,Y 594.34,Z 153.448,A -85,B 0,C 180,E1 -1125.194,E2 -1125.194} C_VEL
LIN {X 0,Y 594.372,Z 153.449,A -85,B 0,C 180,E1 -1127.629,E2 -1127.629} C_VEL
LIN {X 0,Y 594.345,Z 153.448,A -85,B 0,C 180,E1 -1130.321,E2 -1130.321} C_VEL
LIN {X 0,Y 594.365,Z 153.451,A -85,B 0,C 180,E1 -1132.916,E2 -1132.916} C_VEL
LIN {X 0,Y 594.362,Z 153.506,A -85,B 0,C 180,E1 -1134.179,E2 -1134.179} C_VEL
LIN {X 0,Y 594.462,Z 157.93,A -85,B 0,C 180,E1 -1135.85,E2 -1135.85} C_VEL
LIN {X 0,Y 594.472,Z 164.789,A -85,B 0,C 180,E1 -1138.343,E2 -1138.343} C_VEL
LIN {X 0,Y 594.445,Z 172.486,A -85,B 0,C 180,E1 -1141.032,E2 -1141.032} C_VEL
LIN {X 0,Y 594.391,Z 181.175,A -85,B 0,C 180,E1 -1143.977,E2 -1143.977} C_VEL
LIN {X 0,Y 594.365,Z 189.229,A -85,B 0,C 180,E1 -1146.667,E2 -1146.667} C_VEL
LIN {X 0,Y 594.345,Z 198.132,A -85,B 0,C 180,E1 -1149.586,E2 -1149.586} C_VEL
LIN {X 0,Y 594.317,Z 207.036,A -85,B 0,C 180,E1 -1152.451,E2 -1152.451} C_VEL
LIN {X 0,Y 594.286,Z 215.94,A -85,B 0,C 180,E1 -1155.272,E2 -1155.272} C_VEL
LIN {X 0,Y 594.27,Z 224.496,A -85,B 0,C 180,E1 -1157.949,E2 -1157.949} C_VEL
LIN {X 0,Y 594.66,Z 229.301,A -85,B 0,C 180,E1 -1158.043,E2 -1158.043} C_VEL
LIN {X 0,Y 594.605,Z 242.543,A -85,B 0,C 180,E1 -1158.367,E2 -1158.367} C_VEL
LIN {X 0,Y 594.527,Z 254.702,A -85,B 0,C 180,E1 -1158.804,E2 -1158.804} C_VEL
LIN {X 0,Y 594.466,Z 266.233,A -85,B 0,C 180,E1 -1159.356,E2 -1159.356} C_VEL
LIN {X 0,Y 594.451,Z 277.496,A -85,B 0,C 180,E1 -1160.044,E2 -1160.044} C_VEL
LIN {X 0,Y 594.406,Z 287.66,A -85,B 0,C 180,E1 -1160.816,E2 -1160.816} C_VEL
LIN {X 0,Y 594.372,Z 296.797,A -85,B 0,C 180,E1 -1161.673,E2 -1161.673} C_VEL
LIN {X 0,Y 594.316,Z 305.699,A -85,B 0,C 180,E1 -1162.698,E2 -1162.698} C_VEL
LIN {X 0,Y 594.281,Z 312.169,A -85,B 0,C 180,E1 -1163.615,E2 -1163.615} C_VEL
LIN {X 0,Y 594.289,Z 317.685,A -85,B 0,C 180,E1 -1164.572,E2 -1164.572} C_VEL
LIN {X 0,Y 594.27,Z 322.375,A -85,B 0,C 180,E1 -1165.592,E2 -1165.592} C_VEL
LIN {X 0,Y 594.267,Z 325.959,A -85,B 0,C 180,E1 -1166.611,E2 -1166.611} C_VEL
LIN {X 0,Y 594.226,Z 327.81,A -85,B 0,C 180,E1 -1167.289,E2 -1167.289} C_VEL
LIN {X 0,Y 594.242,Z 329.202,A -85,B 0,C 180,E1 -1167.967,E2 -1167.967} C_VEL
LIN {X 0,Y 594.239,Z 330.784,A -85,B 0,C 180,E1 -1169.323,E2 -1169.323} C_VEL
LIN {X 0,Y 594.236,Z 331,A -85,B 0,C 180,E1 -1170,E2 -1170} C_VEL
LIN {X 0,Y 594.247,Z 330.184,A -85,B 0,C 180,E1 -1171.356,E2 -1171.356} C_VEL
LIN {X 0,Y 594.242,Z 329.201,A -85,B 0,C 180,E1 -1172.034,E2 -1172.034} C_VEL
LIN {X 0,Y 594.226,Z 327.809,A -85,B 0,C 180,E1 -1172.712,E2 -1172.712} C_VEL
LIN {X 0,Y 594.289,Z 324.895,A -85,B 0,C 180,E1 -1173.729,E2 -1173.729} C_VEL
LIN {X 0,Y 594.241,Z 320.949,A -85,B 0,C 180,E1 -1174.749,E2 -1174.749} C_VEL
LIN {X 0,Y 594.305,Z 314.877,A -85,B 0,C 180,E1 -1175.939,E2 -1175.939} C_VEL
LIN {X 0,Y 594.308,Z 308.237,A -85,B 0,C 180,E1 -1176.962,E2 -1176.962} C_VEL
LIN {X 0,Y 594.359,Z 299.991,A -85,B 0,C 180,E1 -1177.986,E2 -1177.986} C_VEL
LIN {X 0,Y 594.382,Z 291.539,A -85,B 0,C 180,E1 -1178.842,E2 -1178.842} C_VEL
LIN {X 0,Y 594.43,Z 281.097,A -85,B 0,C 180,E1 -1179.699,E2 -1179.699} C_VEL
LIN {X 0,Y 594.443,Z 270.764,A -85,B 0,C 180,E1 -1180.387,E2 -1180.387} C_VEL
LIN {X 0,Y 594.495,Z 258.801,A -85,B 0,C 180,E1 -1181.018,E2 -1181.018} C_VEL
LIN {X 0,Y 594.556,Z 246.512,A -85,B 0,C 180,E1 -1181.505,E2 -1181.505} C_VEL
LIN {X 0,Y 594.673,Z 233.453,A -85,B 0,C 180,E1 -1181.871,E2 -1181.871} C_VEL
LIN {X 0,Y 594.411,Z 225.641,A -85,B 0,C 180,E1 -1182.028,E2 -1182.028} C_VEL
LIN {X 0,Y 594.275,Z 224.423,A -85,B 0,C 180,E1 -1182.074,E2 -1182.074} C_VEL
LIN {X 0,Y 594.287,Z 214.824,A -85,B 0,C 180,E1 -1185.08,E2 -1185.08} C_VEL
LIN {X 0,Y 594.31,Z 205.92,A -85,B 0,C 180,E1 -1187.905,E2 -1187.905} C_VEL
LIN {X 0,Y 594.346,Z 197.016,A -85,B 0,C 180,E1 -1190.777,E2 -1190.777} C_VEL
LIN {X 0,Y 594.382,Z 188.113,A -85,B 0,C 180,E1 -1193.703,E2 -1193.703} C_VEL
LIN {X 0,Y 594.387,Z 180.272,A -85,B 0,C 180,E1 -1196.323,E2 -1196.323} C_VEL
LIN {X 0,Y 594.42,Z 172.358,A -85,B 0,C 180,E1 -1198.995,E2 -1198.995} C_VEL
LIN {X 0,Y 594.474,Z 164.785,A -85,B 0,C 180,E1 -1201.657,E2 -1201.657} C_VEL
LIN {X 0,Y 594.46,Z 157.93,A -85,B 0,C 180,E1 -1204.149,E2 -1204.149} C_VEL
LIN {X 0,Y 594.53,Z 154.607,A -85,B 0,C 180,E1 -1205.394,E2 -1205.394} C_VEL
LIN {X 0,Y 594.35,Z 153.452,A -85,B 0,C 180,E1 -1205.928,E2 -1205.928} C_VEL
LIN {X 0,Y 594.354,Z 153.451,A -85,B 0,C 180,E1 -1208.805,E2 -1208.805} C_VEL
LIN {X 0,Y 594.37,Z 153.447,A -85,B 0,C 180,E1 -1211.462,E2 -1211.462} C_VEL
LIN {X 0,Y 594.366,Z 153.446,A -85,B 0,C 180,E1 -1214.234,E2 -1214.234} C_VEL
LIN {X 0,Y 594.363,Z 153.45,A -85,B 0,C 180,E1 -1216.7,E2 -1216.7} C_VEL
LIN {X 0,Y 594.34,Z 153.449,A -85,B 0,C 180,E1 -1219.43,E2 -1219.43} C_VEL
LIN {X 0,Y 594.369,Z 153.447,A -85,B 0,C 180,E1 -1222.39,E2 -1222.39} C_VEL
LIN {X 0,Y 594.37,Z 153.445,A -85,B 0,C 180,E1 -1224.669,E2 -1224.669} C_VEL
LIN {X 0,Y 594.36,Z 153.453,A -85,B 0,C 180,E1 -1227.086,E2 -1227.086} C_VEL
LIN {X 0,Y 594.378,Z 153.444,A -85,B 0,C 180,E1 -1229.667,E2 -1229.667} C_VEL
LIN {X 0,Y 594.346,Z 153.45,A -85,B 0,C 180,E1 -1232.538,E2 -1232.538} C_VEL
LIN {X 0,Y 594.348,Z 153.448,A -85,B 0,C 180,E1 -1234.806,E2 -1234.806} C_VEL
LIN {X 0,Y 594.378,Z 153.449,A -85,B 0,C 180,E1 -1237.253,E2 -1237.253} C_VEL
LIN {X 0,Y 594.367,Z 153.446,A -85,B 0,C 180,E1 -1239.946,E2 -1239.946} C_VEL
LIN {X 0,Y 594.369,Z 153.446,A -85,B 0,C 180,E1 -1242.806,E2 -1242.806} C_VEL
LIN {X 0,Y 594.355,Z 153.45,A -85,B 0,C 180,E1 -1245.825,E2 -1245.825} C_VEL
LIN {X 0,Y 594.431,Z 153.445,A -85,B 0,C 180,E1 -1248.887,E2 -1248.887} C_VEL
LIN {X 0,Y 594.404,Z 153.442,A -85,B 0,C 180,E1 -1251.843,E2 -1251.843} C_VEL
LIN {X 0,Y 594.381,Z 153.444,A -85,B 0,C 180,E1 -1254.572,E2 -1254.572} C_VEL
LIN {X 0,Y 594.396,Z 153.449,A -85,B 0,C 180,E1 -1257.289,E2 -1257.289} C_VEL
LIN {X 0,Y 594.37,Z 153.445,A -85,B 0,C 180,E1 -1260,E2 -1260} C_VEL
LIN {X 0,Y 594.404,Z 153.443,A -85,B 0,C 180,E1 -1262.711,E2 -1262.711} C_VEL
LIN {X 0,Y 594.389,Z 153.446,A -85,B 0,C 180,E1 -1265.428,E2 -1265.428} C_VEL
LIN {X 0,Y 594.394,Z 153.442,A -85,B 0,C 180,E1 -1268.157,E2 -1268.157} C_VEL
LIN {X 0,Y 594.372,Z 153.448,A -85,B 0,C 180,E1 -1271.083,E2 -1271.083} C_VEL
LIN {X 0,Y 594.382,Z 153.45,A -85,B 0,C 180,E1 -1274.185,E2 -1274.185} C_VEL
LIN {X 0,Y 594.351,Z 153.449,A -85,B 0,C 180,E1 -1275.356,E2 -1275.356} C_VEL
LIN {X 0,Y 593.688,Z 153.536,A -85,B 0,C 180,E1 -1275.921,E2 -1275.921} C_VEL
LIN {X 0,Y 590.833,Z 153.89,A -85,B 0,C 180,E1 -1276.84,E2 -1276.84} C_VEL
LIN {X 0,Y 588.424,Z 154.192,A -85,B 0,C 180,E1 -1277.578,E2 -1277.578} C_VEL
LIN {X 0,Y 587.397,Z 154.314,A -85,B 0,C 180,E1 -1278.148,E2 -1278.148} C_VEL
LIN {X 0,Y 587.317,Z 154.323,A -85,B 0,C 180,E1 -1278.341,E2 -1278.341} C_VEL
LIN {X 0,Y 587.329,Z 154.327,A -85,B 0,C 180,E1 -1281.046,E2 -1281.046} C_VEL
LIN {X 0,Y 587.302,Z 154.326,A -85,B 0,C 180,E1 -1283.26,E2 -1283.26} C_VEL
LIN {X 0,Y 587.336,Z 154.325,A -85,B 0,C 180,E1 -1286.184,E2 -1286.184} C_VEL
LIN {X 0,Y 587.333,Z 154.327,A -85,B 0,C 180,E1 -1289.137,E2 -1289.137} C_VEL
LIN {X 0,Y 587.342,Z 154.32,A -85,B 0,C 180,E1 -1291.841,E2 -1291.841} C_VEL
LIN {X 0,Y 587.331,Z 154.329,A -85,B 0,C 180,E1 -1294.351,E2 -1294.351} C_VEL
LIN {X 0,Y 587.328,Z 154.322,A -85,B 0,C 180,E1 -1296.749,E2 -1296.749} C_VEL
LIN {X 0,Y 587.327,Z 154.33,A -85,B 0,C 180,E1 -1299.361,E2 -1299.361} C_VEL
LIN {X 0,Y 587.319,Z 154.323,A -85,B 0,C 180,E1 -1302.11,E2 -1302.11} C_VEL
LIN {X 0,Y 587.302,Z 154.326,A -85,B 0,C 180,E1 -1305.091,E2 -1305.091} C_VEL
LIN {X 0,Y 587.342,Z 154.326,A -85,B 0,C 180,E1 -1307.93,E2 -1307.93} C_VEL
LIN {X 0,Y 587.302,Z 154.332,A -85,B 0,C 180,E1 -1311.063,E2 -1311.063} C_VEL
LIN {X 0,Y 587.309,Z 154.327,A -85,B 0,C 180,E1 -1312.392,E2 -1312.392} C_VEL
LIN {X 0,Y 587.299,Z 155.35,A -85,B 0,C 180,E1 -1313.3,E2 -1313.3} C_VEL
LIN {X 0,Y 587.269,Z 159.526,A -85,B 0,C 180,E1 -1315.776,E2 -1315.776} C_VEL
LIN {X 0,Y 587.292,Z 163.708,A -85,B 0,C 180,E1 -1318.23,E2 -1318.23} C_VEL
LIN {X 0,Y 587.247,Z 168.344,A -85,B 0,C 180,E1 -1320.886,E2 -1320.886} C_VEL
LIN {X 0,Y 587.224,Z 172.004,A -85,B 0,C 180,E1 -1322.95,E2 -1322.95} C_VEL
LIN {X 0,Y 587.2,Z 176.519,A -85,B 0,C 180,E1 -1325.454,E2 -1325.454} C_VEL
LIN {X 0,Y 587.172,Z 181.723,A -85,B 0,C 180,E1 -1328.221,E2 -1328.221} C_VEL
LIN {X 0,Y 587.193,Z 187.32,A -85,B 0,C 180,E1 -1331.147,E2 -1331.147} C_VEL
LIN {X 0,Y 587.145,Z 192.906,A -85,B 0,C 180,E1 -1334.021,E2 -1334.021} C_VEL
LIN {X 0,Y 587.161,Z 196.738,A -85,B 0,C 180,E1 -1335.884,E2 -1335.884} C_VEL
LIN {X 0,Y 587.725,Z 201.995,A -85,B 0,C 180,E1 -1335.998,E2 -1335.998} C_VEL
LIN {X 0,Y 587.661,Z 214.582,A -85,B 0,C 180,E1 -1336.338,E2 -1336.338} C_VEL
LIN {X 0,Y 587.551,Z 226.117,A -85,B 0,C 180,E1 -1336.776,E2 -1336.776} C_VEL
LIN {X 0,Y 587.43,Z 238.331,A -85,B 0,C 180,E1 -1337.389,E2 -1337.389} C_VEL
LIN {X 0,Y 587.459,Z 249.231,A -85,B 0,C 180,E1 -1338.091,E2 -1338.091} C_VEL
LIN {X 0,Y 587.345,Z 260.052,A -85,B 0,C 180,E1 -1338.963,E2 -1338.963} C_VEL
LIN {X 0,Y 587.303,Z 268.836,A -85,B 0,C 180,E1 -1339.834,E2 -1339.834} C_VEL
LIN {X 0,Y 587.259,Z 277.359,A -85,B 0,C 180,E1 -1340.876,E2 -1340.876} C_VEL
LIN {X 0,Y 587.213,Z 284.187,A -85,B 0,C 180,E1 -1341.916,E2 -1341.916} C_VEL
LIN {X 0,Y 587.211,Z 290.448,A -85,B 0,C 180,E1 -1343.126,E2 -1343.126} C_VEL
LIN {X 0,Y 587.179,Z 294.518,A -85,B 0,C 180,E1 -1344.161,E2 -1344.161} C_VEL
LIN {X 0,Y 587.131,Z 297.536,A -85,B 0,C 180,E1 -1345.193,E2 -1345.193} C_VEL
LIN {X 0,Y 587.171,Z 299.026,A -85,B 0,C 180,E1 -1345.882,E2 -1345.882} C_VEL
LIN {X 0,Y 587.182,Z 300.066,A -85,B 0,C 180,E1 -1346.569,E2 -1346.569} C_VEL
LIN {X 0,Y 587.14,Z 300.983,A -85,B 0,C 180,E1 -1347.942,E2 -1347.942} C_VEL
LIN {X 0,Y 587.147,Z 300.854,A -85,B 0,C 180,E1 -1348.628,E2 -1348.628} C_VEL
LIN {X 0,Y 587.139,Z 299.368,A -85,B 0,C 180,E1 -1350,E2 -1350} C_VEL
LIN {X 0,Y 587.14,Z 298.038,A -85,B 0,C 180,E1 -1350.685,E2 -1350.685} C_VEL
LIN {X 0,Y 587.18,Z 295.223,A -85,B 0,C 180,E1 -1351.714,E2 -1351.714} C_VEL
LIN {X 0,Y 587.153,Z 291.395,A -85,B 0,C 180,E1 -1352.744,E2 -1352.744} C_VEL
LIN {X 0,Y 587.214,Z 286.448,A -85,B 0,C 180,E1 -1353.774,E2 -1353.774} C_VEL
LIN {X 0,Y 587.28,Z 280.237,A -85,B 0,C 180,E1 -1354.804,E2 -1354.804} C_VEL
LIN {X 0,Y 587.266,Z 272.491,A -85,B 0,C 180,E1 -1355.837,E2 -1355.837} C_VEL
LIN {X 0,Y 587.335,Z 262.815,A -85,B 0,C 180,E1 -1356.871,E2 -1356.871} C_VEL
LIN {X 0,Y 587.416,Z 252.792,A -85,B 0,C 180,E1 -1357.734,E2 -1357.734} C_VEL
LIN {X 0,Y 587.449,Z 241.479,A -85,B 0,C 180,E1 -1358.513,E2 -1358.513} C_VEL
LIN {X 0,Y 587.528,Z 230.38,A -85,B 0,C 180,E1 -1359.118,E2 -1359.118} C_VEL
LIN {X 0,Y 587.644,Z 217.977,A -85,B 0,C 180,E1 -1359.638,E2 -1359.638} C_VEL
LIN {X 0,Y 587.726,Z 204.746,A -85,B 0,C 180,E1 -1360.027,E2 -1360.027} C_VEL
LIN {X 0,Y 587.44,Z 198.673,A -85,B 0,C 180,E1 -1360.163,E2 -1360.163} C_VEL
LIN {X 0,Y 587.113,Z 196.555,A -85,B 0,C 180,E1 -1360.212,E2 -1360.212} C_VEL
LIN {X 0,Y 587.151,Z 192.18,A -85,B 0,C 180,E1 -1362.441,E2 -1362.441} C_VEL
LIN {X 0,Y 587.163,Z 186.699,A -85,B 0,C 180,E1 -1365.266,E2 -1365.266} C_VEL
LIN {X 0,Y 587.209,Z 182.595,A -85,B 0,C 180,E1 -1367.408,E2 -1367.408} C_VEL
LIN {X 0,Y 587.195,Z 178.497,A -85,B 0,C 180,E1 -1369.578,E2 -1369.578} C_VEL
LIN {X 0,Y 587.209,Z 174.433,A -85,B 0,C 180,E1 -1371.777,E2 -1371.777} C_VEL
LIN {X 0,Y 587.243,Z 169.496,A -85,B 0,C 180,E1 -1374.555,E2 -1374.555} C_VEL
LIN {X 0,Y 587.241,Z 165.139,A -85,B 0,C 180,E1 -1377.048,E2 -1377.048} C_VEL
LIN {X 0,Y 587.257,Z 161.105,A -85,B 0,C 180,E1 -1379.382,E2 -1379.382} C_VEL
LIN {X 0,Y 587.303,Z 156.951,A -85,B 0,C 180,E1 -1381.828,E2 -1381.828} C_VEL
LIN {X 0,Y 587.247,Z 154.338,A -85,B 0,C 180,E1 -1383.399,E2 -1383.399} C_VEL
LIN {X 0,Y 587.282,Z 154.329,A -85,B 0,C 180,E1 -1385.535,E2 -1385.535} C_VEL
LIN {X 0,Y 587.309,Z 154.331,A -85,B 0,C 180,E1 -1388.477,E2 -1388.477} C_VEL
LIN {X 0,Y 587.323,Z 154.322,A -85,B 0,C 180,E1 -1391.154,E2 -1391.154} C_VEL
LIN {X 0,Y 587.316,Z 154.328,A -85,B 0,C 180,E1 -1393.947,E2 -1393.947} C_VEL
LIN {X 0,Y 587.317,Z 154.328,A -85,B 0,C 180,E1 -1396.993,E2 -1396.993} C_VEL
LIN {X 0,Y 587.299,Z 154.325,A -85,B 0,C 180,E1 -1399.744,E2 -1399.744} C_VEL
LIN {X 0,Y 587.317,Z 154.33,A -85,B 0,C 180,E1 -1402.39,E2 -1402.39} C_VEL
LIN {X 0,Y 587.295,Z 154.326,A -85,B 0,C 180,E1 -1404.942,E2 -1404.942} C_VEL
LIN {X 0,Y 587.319,Z 154.327,A -85,B 0,C 180,E1 -1407.419,E2 -1407.419} C_VEL
LIN {X 0,Y 587.324,Z 154.324,A -85,B 0,C 180,E1 -1409.829,E2 -1409.829} C_VEL
LIN {X 0,Y 587.327,Z 154.322,A -85,B 0,C 180,E1 -1412.303,E2 -1412.303} C_VEL
LIN {X 0,Y 587.324,Z 154.328,A -85,B 0,C 180,E1 -1414.483,E2 -1414.483} C_VEL
LIN {X 0,Y 587.339,Z 154.321,A -85,B 0,C 180,E1 -1417.486,E2 -1417.486} C_VEL
LIN {X 0,Y 587.309,Z 154.325,A -85,B 0,C 180,E1 -1420.423,E2 -1420.423} C_VEL
LIN {X 0,Y 587.344,Z 154.327,A -85,B 0,C 180,E1 -1423.311,E2 -1423.311} C_VEL
LIN {X 0,Y 587.338,Z 154.321,A -85,B 0,C 180,E1 -1426.154,E2 -1426.154} C_VEL
LIN {X 0,Y 587.37,Z 154.319,A -85,B 0,C 180,E1 -1428.963,E2 -1428.963} C_VEL
LIN {X 0,Y 587.352,Z 154.322,A -85,B 0,C 180,E1 -1431.744,E2 -1431.744} C_VEL
LIN {X 0,Y 587.34,Z 154.32,A -85,B 0,C 180,E1 -1434.507,E2 -1434.507} C_VEL
LIN {X 0,Y 587.356,Z 154.325,A -85,B 0,C 180,E1 -1437.256,E2 -1437.256} C_VEL
LIN {X 0,Y 587.331,Z 154.321,A -85,B 0,C 180,E1 -1440,E2 -1440} C_VEL
LIN {X 0,Y 587.366,Z 154.322,A -85,B 0,C 180,E1 -1442.743,E2 -1442.743} C_VEL
LIN {X 0,Y 587.347,Z 154.321,A -85,B 0,C 180,E1 -1445.493,E2 -1445.493} C_VEL
LIN {X 0,Y 587.352,Z 154.32,A -85,B 0,C 180,E1 -1448.255,E2 -1448.255} C_VEL
LIN {X 0,Y 587.388,Z 154.321,A -85,B 0,C 180,E1 -1451.176,E2 -1451.176} C_VEL
LIN {X 0,Y 587.339,Z 154.322,A -85,B 0,C 180,E1 -1454.268,E2 -1454.268} C_VEL
LIN {X 0,Y 587.319,Z 154.323,A -85,B 0,C 180,E1 -1457.407,E2 -1457.407} C_VEL
LIN {X 0,Y 587.308,Z 154.327,A -85,B 0,C 180,E1 -1460.306,E2 -1460.306} C_VEL
LIN {X 0,Y 587.35,Z 154.324,A -85,B 0,C 180,E1 -1463.258,E2 -1463.258} C_VEL
LIN {X 0,Y 587.338,Z 154.32,A -85,B 0,C 180,E1 -1466.186,E2 -1466.186} C_VEL
LIN {X 0,Y 587.347,Z 154.321,A -85,B 0,C 180,E1 -1469.141,E2 -1469.141} C_VEL
LIN {X 0,Y 587.328,Z 154.325,A -85,B 0,C 180,E1 -1471.841,E2 -1471.841} C_VEL
LIN {X 0,Y 587.315,Z 154.326,A -85,B 0,C 180,E1 -1474.35,E2 -1474.35} C_VEL
LIN {X 0,Y 587.324,Z 154.323,A -85,B 0,C 180,E1 -1476.749,E2 -1476.749} C_VEL
LIN {X 0,Y 587.33,Z 154.326,A -85,B 0,C 180,E1 -1479.361,E2 -1479.361} C_VEL
LIN {X 0,Y 587.342,Z 154.321,A -85,B 0,C 180,E1 -1482.114,E2 -1482.114} C_VEL
LIN {X 0,Y 587.293,Z 154.326,A -85,B 0,C 180,E1 -1485.091,E2 -1485.091} C_VEL
LIN {X 0,Y 587.333,Z 154.329,A -85,B 0,C 180,E1 -1487.93,E2 -1487.93} C_VEL
LIN {X 0,Y 587.305,Z 154.326,A -85,B 0,C 180,E1 -1490.641,E2 -1490.641} C_VEL
LIN {X 0,Y 587.331,Z 154.328,A -85,B 0,C 180,E1 -1493.295,E2 -1493.295} C_VEL
LIN {X 0,Y 587.335,Z 154.427,A -85,B 0,C 180,E1 -1494.054,E2 -1494.054} C_VEL
LIN {X 0,Y 587.504,Z 158.536,A -85,B 0,C 180,E1 -1495.63,E2 -1495.63} C_VEL
LIN {X 0,Y 587.468,Z 165.626,A -85,B 0,C 180,E1 -1498.242,E2 -1498.242} C_VEL
LIN {X 0,Y 587.441,Z 172.993,A -85,B 0,C 180,E1 -1500.851,E2 -1500.851} C_VEL
LIN {X 0,Y 587.36,Z 181.624,A -85,B 0,C 180,E1 -1503.819,E2 -1503.819} C_VEL
LIN {X 0,Y 587.331,Z 189.229,A -85,B 0,C 180,E1 -1506.37,E2 -1506.37} C_VEL
LIN {X 0,Y 587.288,Z 198.148,A -85,B 0,C 180,E1 -1509.335,E2 -1509.335} C_VEL
LIN {X 0,Y 587.267,Z 207.036,A -85,B 0,C 180,E1 -1512.234,E2 -1512.234} C_VEL
LIN {X 0,Y 587.21,Z 215.94,A -85,B 0,C 180,E1 -1515.09,E2 -1515.09} C_VEL
LIN {X 0,Y 587.161,Z 224.496,A -85,B 0,C 180,E1 -1517.801,E2 -1517.801} C_VEL
LIN {X 0,Y 587.738,Z 229.301,A -85,B 0,C 180,E1 -1517.9,E2 -1517.9} C_VEL
LIN {X 0,Y 587.673,Z 242.544,A -85,B 0,C 180,E1 -1518.227,E2 -1518.227} C_VEL
LIN {X 0,Y 587.561,Z 254.505,A -85,B 0,C 180,E1 -1518.66,E2 -1518.66} C_VEL
LIN {X 0,Y 587.484,Z 266.234,A -85,B 0,C 180,E1 -1519.228,E2 -1519.228} C_VEL
LIN {X 0,Y 587.444,Z 277.497,A -85,B 0,C 180,E1 -1519.924,E2 -1519.924} C_VEL
LIN {X 0,Y 587.384,Z 287.66,A -85,B 0,C 180,E1 -1520.706,E2 -1520.706} C_VEL
LIN {X 0,Y 587.339,Z 296.797,A -85,B 0,C 180,E1 -1521.572,E2 -1521.572} C_VEL
LIN {X 0,Y 587.258,Z 305.698,A -85,B 0,C 180,E1 -1522.609,E2 -1522.609} C_VEL
LIN {X 0,Y 587.195,Z 312.746,A -85,B 0,C 180,E1 -1523.627,E2 -1523.627} C_VEL
LIN {X 0,Y 587.211,Z 317.685,A -85,B 0,C 180,E1 -1524.507,E2 -1524.507} C_VEL
LIN {X 0,Y 587.188,Z 322.375,A -85,B 0,C 180,E1 -1525.539,E2 -1525.539} C_VEL
LIN {X 0,Y 587.193,Z 325.959,A -85,B 0,C 180,E1 -1526.57,E2 -1526.57} C_VEL
LIN {X 0,Y 587.132,Z 327.81,A -85,B 0,C 180,E1 -1527.256,E2 -1527.256} C_VEL
LIN {X 0,Y 587.141,Z 329.201,A -85,B 0,C 180,E1 -1527.943,E2 -1527.943} C_VEL
LIN {X 0,Y 587.14,Z 330.785,A -85,B 0,C 180,E1 -1529.315,E2 -1529.315} C_VEL
LIN {X 0,Y 587.137,Z 331,A -85,B 0,C 180,E1 -1530,E2 -1530} C_VEL
LIN {X 0,Y 587.147,Z 330.185,A -85,B 0,C 180,E1 -1531.372,E2 -1531.372} C_VEL
LIN {X 0,Y 587.141,Z 329.2,A -85,B 0,C 180,E1 -1532.058,E2 -1532.058} C_VEL
LIN {X 0,Y 587.132,Z 327.809,A -85,B 0,C 180,E1 -1532.745,E2 -1532.745} C_VEL
LIN {X 0,Y 587.213,Z 324.895,A -85,B 0,C 180,E1 -1533.774,E2 -1533.774} C_VEL
LIN {X 0,Y 587.147,Z 320.949,A -85,B 0,C 180,E1 -1534.806,E2 -1534.806} C_VEL
LIN {X 0,Y 587.218,Z 314.877,A -85,B 0,C 180,E1 -1536.011,E2 -1536.011} C_VEL
LIN {X 0,Y 587.245,Z 308.237,A -85,B 0,C 180,E1 -1537.046,E2 -1537.046} C_VEL
LIN {X 0,Y 587.299,Z 299.991,A -85,B 0,C 180,E1 -1538.083,E2 -1538.083} C_VEL
LIN {X 0,Y 587.343,Z 291.54,A -85,B 0,C 180,E1 -1538.949,E2 -1538.949} C_VEL
LIN {X 0,Y 587.418,Z 281.099,A -85,B 0,C 180,E1 -1539.816,E2 -1539.816} C_VEL
LIN {X 0,Y 587.445,Z 270.762,A -85,B 0,C 180,E1 -1540.512,E2 -1540.512} C_VEL
LIN {X 0,Y 587.527,Z 259.19,A -85,B 0,C 180,E1 -1541.132,E2 -1541.132} C_VEL
LIN {X 0,Y 587.618,Z 246.716,A -85,B 0,C 180,E1 -1541.636,E2 -1541.636} C_VEL
LIN {X 0,Y 587.738,Z 233.452,A -85,B 0,C 180,E1 -1542.013,E2 -1542.013} C_VEL
LIN {X 0,Y 587.52,Z 226.673,A -85,B 0,C 180,E1 -1542.154,E2 -1542.154} C_VEL
LIN {X 0,Y 587.161,Z 224.423,A -85,B 0,C 180,E1 -1542.222,E2 -1542.222} C_VEL
LIN {X 0,Y 587.211,Z 215.937,A -85,B 0,C 180,E1 -1544.911,E2 -1544.911} C_VEL
LIN {X 0,Y 587.267,Z 207.033,A -85,B 0,C 180,E1 -1547.767,E2 -1547.767} C_VEL
LIN {X 0,Y 587.289,Z 198.145,A -85,B 0,C 180,E1 -1550.666,E2 -1550.666} C_VEL
LIN {X 0,Y 587.332,Z 189.226,A -85,B 0,C 180,E1 -1553.631,E2 -1553.631} C_VEL
LIN {X 0,Y 587.366,Z 181.316,A -85,B 0,C 180,E1 -1556.276,E2 -1556.276} C_VEL
LIN {X 0,Y 587.389,Z 172.975,A -85,B 0,C 180,E1 -1559.14,E2 -1559.14} C_VEL
LIN {X 0,Y 587.465,Z 165.356,A -85,B 0,C 180,E1 -1561.854,E2 -1561.854} C_VEL
LIN {X 0,Y 587.48,Z 158.554,A -85,B 0,C 180,E1 -1564.366,E2 -1564.366} C_VEL
LIN {X 0,Y 587.314,Z 154.33,A -85,B 0,C 180,E1 -1566.002,E2 -1566.002} C_VEL
LIN {X 0,Y 587.304,Z 154.333,A -85,B 0,C 180,E1 -1568.479,E2 -1568.479} C_VEL
LIN {X 0,Y 587.326,Z 154.323,A -85,B 0,C 180,E1 -1571.155,E2 -1571.155} C_VEL
LIN {X 0,Y 587.319,Z 154.325,A -85,B 0,C 180,E1 -1573.947,E2 -1573.947} C_VEL
LIN {X 0,Y 587.305,Z 154.332,A -85,B 0,C 180,E1 -1576.993,E2 -1576.993} C_VEL
LIN {X 0,Y 587.293,Z 154.328,A -85,B 0,C 180,E1 -1579.744,E2 -1579.744} C_VEL
LIN {X 0,Y 587.324,Z 154.325,A -85,B 0,C 180,E1 -1582.391,E2 -1582.391} C_VEL
LIN {X 0,Y 587.336,Z 154.323,A -85,B 0,C 180,E1 -1584.945,E2 -1584.945} C_VEL
LIN {X 0,Y 587.322,Z 154.325,A -85,B 0,C 180,E1 -1587.42,E2 -1587.42} C_VEL
LIN {X 0,Y 587.325,Z 154.323,A -85,B 0,C 180,E1 -1589.829,E2 -1589.829} C_VEL
LIN {X 0,Y 587.324,Z 154.327,A -85,B 0,C 180,E1 -1592.305,E2 -1592.305} C_VEL
LIN {X 0,Y 587.324,Z 154.327,A -85,B 0,C 180,E1 -1595.24,E2 -1595.24} C_VEL
LIN {X 0,Y 587.347,Z 154.322,A -85,B 0,C 180,E1 -1597.487,E2 -1597.487} C_VEL
LIN {X 0,Y 587.33,Z 154.328,A -85,B 0,C 180,E1 -1600.425,E2 -1600.425} C_VEL
LIN {X 0,Y 587.337,Z 154.322,A -85,B 0,C 180,E1 -1603.311,E2 -1603.311} C_VEL
LIN {X 0,Y 587.325,Z 154.323,A -85,B 0,C 180,E1 -1606.154,E2 -1606.154} C_VEL
LIN {X 0,Y 587.379,Z 154.322,A -85,B 0,C 180,E1 -1608.963,E2 -1608.963} C_VEL
LIN {X 0,Y 587.355,Z 154.319,A -85,B 0,C 180,E1 -1611.745,E2 -1611.745} C_VEL
LIN {X 0,Y 587.341,Z 154.326,A -85,B 0,C 180,E1 -1613.818,E2 -1613.818} C_VEL
LIN {X 0,Y 587.296,Z 154.33,A -85,B 0,C 180,E1 -1615.883,E2 -1615.883} C_VEL
LIN {X 0,Y 587.324,Z 154.323,A -85,B 0,C 180,E1 -1617.943,E2 -1617.943} C_VEL
LIN {X 0,Y 587.381,Z 154.322,A -85,B 0,C 180,E1 -1620.686,E2 -1620.686} C_VEL
LIN {X 0,Y 587.322,Z 154.323,A -85,B 0,C 180,E1 -1623.43,E2 -1623.43} C_VEL
LIN {X 0,Y 587.333,Z 154.323,A -85,B 0,C 180,E1 -1626.183,E2 -1626.183} C_VEL
LIN {X 0,Y 587.329,Z 154.328,A -85,B 0,C 180,E1 -1628.949,E2 -1628.949} C_VEL
LIN {X 0,Y 587.308,Z 154.325,A -85,B 0,C 180,E1 -1631.738,E2 -1631.738} C_VEL
LIN {X 0,Y 587.321,Z 154.325,A -85,B 0,C 180,E1 -1634.554,E2 -1634.554} C_VEL
LIN {X 0,Y 587.341,Z 154.326,A -85,B 0,C 180,E1 -1637.407,E2 -1637.407} C_VEL
LIN {X 0,Y 587.317,Z 154.323,A -85,B 0,C 180,E1 -1638.341,E2 -1638.341} C_VEL
LIN {X 0,Y 586.664,Z 154.409,A -85,B 0,C 180,E1 -1638.914,E2 -1638.914} C_VEL
LIN {X 0,Y 583.823,Z 154.763,A -85,B 0,C 180,E1 -1639.842,E2 -1639.842} C_VEL
LIN {X 0,Y 581.406,Z 155.065,A -85,B 0,C 180,E1 -1640.589,E2 -1640.589} C_VEL
LIN {X 0,Y 580.355,Z 155.195,A -85,B 0,C 180,E1 -1641.165,E2 -1641.165} C_VEL
LIN {X 0,Y 580.263,Z 155.204,A -85,B 0,C 180,E1 -1641.36,E2 -1641.36} C_VEL
LIN {X 0,Y 580.257,Z 155.204,A -85,B 0,C 180,E1 -1643.559,E2 -1643.559} C_VEL
LIN {X 0,Y 580.302,Z 155.199,A -85,B 0,C 180,E1 -1646.343,E2 -1646.343} C_VEL
LIN {X 0,Y 580.288,Z 155.206,A -85,B 0,C 180,E1 -1649.314,E2 -1649.314} C_VEL
LIN {X 0,Y 580.287,Z 155.201,A -85,B 0,C 180,E1 -1652.202,E2 -1652.202} C_VEL
LIN {X 0,Y 580.271,Z 155.204,A -85,B 0,C 180,E1 -1654.698,E2 -1654.698} C_VEL
LIN {X 0,Y 580.276,Z 155.203,A -85,B 0,C 180,E1 -1657.271,E2 -1657.271} C_VEL
LIN {X 0,Y 580.281,Z 155.2,A -85,B 0,C 180,E1 -1660.273,E2 -1660.273} C_VEL
LIN {X 0,Y 580.268,Z 155.208,A -85,B 0,C 180,E1 -1662.708,E2 -1662.708} C_VEL
LIN {X 0,Y 580.256,Z 155.204,A -85,B 0,C 180,E1 -1665.611,E2 -1665.611} C_VEL
LIN {X 0,Y 580.285,Z 155.201,A -85,B 0,C 180,E1 -1668.235,E2 -1668.235} C_VEL
LIN {X 0,Y 580.258,Z 155.208,A -85,B 0,C 180,E1 -1670.966,E2 -1670.966} C_VEL
LIN {X 0,Y 580.232,Z 155.272,A -85,B 0,C 180,E1 -1672.729,E2 -1672.729} C_VEL
LIN {X 0,Y 580.212,Z 159.8,A -85,B 0,C 180,E1 -1675.455,E2 -1675.455} C_VEL
LIN {X 0,Y 580.231,Z 164.067,A -85,B 0,C 180,E1 -1677.982,E2 -1677.982} C_VEL
LIN {X 0,Y 580.178,Z 168.745,A -85,B 0,C 180,E1 -1680.713,E2 -1680.713} C_VEL
LIN {X 0,Y 580.175,Z 172.049,A -85,B 0,C 180,E1 -1682.594,E2 -1682.594} C_VEL
LIN {X 0,Y 580.149,Z 176.845,A -85,B 0,C 180,E1 -1685.308,E2 -1685.308} C_VEL
LIN {X 0,Y 580.087,Z 181.671,A -85,B 0,C 180,E1 -1687.941,E2 -1687.941} C_VEL
LIN {X 0,Y 580.099,Z 187.27,A -85,B 0,C 180,E1 -1690.908,E2 -1690.908} C_VEL
LIN {X 0,Y 580.065,Z 192.857,A -85,B 0,C 180,E1 -1693.82,E2 -1693.82} C_VEL
LIN {X 0,Y 580.053,Z 196.587,A -85,B 0,C 180,E1 -1695.73,E2 -1695.73} C_VEL
LIN {X 0,Y 580.784,Z 203.306,A -85,B 0,C 180,E1 -1695.883,E2 -1695.883} C_VEL
LIN {X 0,Y 580.695,Z 216.474,A -85,B 0,C 180,E1 -1696.261,E2 -1696.261} C_VEL
LIN {X 0,Y 580.585,Z 227.555,A -85,B 0,C 180,E1 -1696.704,E2 -1696.704} C_VEL
LIN {X 0,Y 580.429,Z 239.442,A -85,B 0,C 180,E1 -1697.323,E2 -1697.323} C_VEL
LIN {X 0,Y 580.406,Z 251.26,A -85,B 0,C 180,E1 -1698.121,E2 -1698.121} C_VEL
LIN {X 0,Y 580.3,Z 261.23,A -85,B 0,C 180,E1 -1698.958,E2 -1698.958} C_VEL
LIN {X 0,Y 580.248,Z 270.179,A -85,B 0,C 180,E1 -1699.885,E2 -1699.885} C_VEL
LIN {X 0,Y 580.173,Z 278.429,A -85,B 0,C 180,E1 -1700.94,E2 -1700.94} C_VEL
LIN {X 0,Y 580.142,Z 285.06,A -85,B 0,C 180,E1 -1701.992,E2 -1701.992} C_VEL
LIN {X 0,Y 580.142,Z 290.337,A -85,B 0,C 180,E1 -1703.042,E2 -1703.042} C_VEL
LIN {X 0,Y 580.094,Z 294.434,A -85,B 0,C 180,E1 -1704.089,E2 -1704.089} C_VEL
LIN {X 0,Y 580.035,Z 297.476,A -85,B 0,C 180,E1 -1705.134,E2 -1705.134} C_VEL
LIN {X 0,Y 580.089,Z 298.982,A -85,B 0,C 180,E1 -1705.831,E2 -1705.831} C_VEL
LIN {X 0,Y 580.107,Z 300.038,A -85,B 0,C 180,E1 -1706.527,E2 -1706.527} C_VEL
LIN {X 0,Y 580.039,Z 300.977,A -85,B 0,C 180,E1 -1707.917,E2 -1707.917} C_VEL
LIN {X 0,Y 580.046,Z 300.868,A -85,B 0,C 180,E1 -1708.611,E2 -1708.611} C_VEL
LIN {X 0,Y 580.04,Z 299.406,A -85,B 0,C 180,E1 -1710,E2 -1710} C_VEL
LIN {X 0,Y 580.041,Z 298.087,A -85,B 0,C 180,E1 -1710.694,E2 -1710.694} C_VEL
LIN {X 0,Y 580.086,Z 295.296,A -85,B 0,C 180,E1 -1711.735,E2 -1711.735} C_VEL
LIN {X 0,Y 580.066,Z 291.493,A -85,B 0,C 180,E1 -1712.777,E2 -1712.777} C_VEL
LIN {X 0,Y 580.141,Z 286.573,A -85,B 0,C 180,E1 -1713.82,E2 -1713.82} C_VEL
LIN {X 0,Y 580.206,Z 280.392,A -85,B 0,C 180,E1 -1714.863,E2 -1714.863} C_VEL
LIN {X 0,Y 580.209,Z 272.695,A -85,B 0,C 180,E1 -1715.909,E2 -1715.909} C_VEL
LIN {X 0,Y 580.297,Z 264.25,A -85,B 0,C 180,E1 -1716.838,E2 -1716.838} C_VEL
LIN {X 0,Y 580.37,Z 254.186,A -85,B 0,C 180,E1 -1717.741,E2 -1717.741} C_VEL
LIN {X 0,Y 580.444,Z 243.273,A -85,B 0,C 180,E1 -1718.529,E2 -1718.529} C_VEL
LIN {X 0,Y 580.511,Z 232.611,A -85,B 0,C 180,E1 -1719.142,E2 -1719.142} C_VEL
LIN {X 0,Y 580.641,Z 219.784,A -85,B 0,C 180,E1 -1719.711,E2 -1719.711} C_VEL
LIN {X 0,Y 580.76,Z 206.658,A -85,B 0,C 180,E1 -1720.127,E2 -1720.127} C_VEL
LIN {X 0,Y 580.554,Z 199.913,A -85,B 0,C 180,E1 -1720.285,E2 -1720.285} C_VEL
LIN {X 0,Y 580.033,Z 196.518,A -85,B 0,C 180,E1 -1720.382,E2 -1720.382} C_VEL
LIN {X 0,Y 580.07,Z 192.229,A -85,B 0,C 180,E1 -1722.595,E2 -1722.595} C_VEL
LIN {X 0,Y 580.097,Z 186.749,A -85,B 0,C 180,E1 -1725.457,E2 -1725.457} C_VEL
LIN {X 0,Y 580.119,Z 182.645,A -85,B 0,C 180,E1 -1727.628,E2 -1727.628} C_VEL
LIN {X 0,Y 580.103,Z 178.561,A -85,B 0,C 180,E1 -1729.827,E2 -1729.827} C_VEL
LIN {X 0,Y 580.167,Z 174.582,A -85,B 0,C 180,E1 -1732.055,E2 -1732.055} C_VEL
LIN {X 0,Y 580.174,Z 169.289,A -85,B 0,C 180,E1 -1735.083,E2 -1735.083} C_VEL
LIN {X 0,Y 580.214,Z 164.515,A -85,B 0,C 180,E1 -1737.842,E2 -1737.842} C_VEL
LIN {X 0,Y 580.224,Z 159.705,A -85,B 0,C 180,E1 -1740.683,E2 -1740.683} C_VEL
LIN {X 0,Y 580.214,Z 155.33,A -85,B 0,C 180,E1 -1743.302,E2 -1743.302} C_VEL
LIN {X 0,Y 580.236,Z 155.206,A -85,B 0,C 180,E1 -1745.545,E2 -1745.545} C_VEL
LIN {X 0,Y 580.27,Z 155.204,A -85,B 0,C 180,E1 -1748.144,E2 -1748.144} C_VEL
LIN {X 0,Y 580.287,Z 155.2,A -85,B 0,C 180,E1 -1750.84,E2 -1750.84} C_VEL
LIN {X 0,Y 580.272,Z 155.208,A -85,B 0,C 180,E1 -1753.654,E2 -1753.654} C_VEL
LIN {X 0,Y 580.272,Z 155.201,A -85,B 0,C 180,E1 -1756.605,E2 -1756.605} C_VEL
LIN {X 0,Y 580.296,Z 155.202,A -85,B 0,C 180,E1 -1759.156,E2 -1759.156} C_VEL
LIN {X 0,Y 580.264,Z 155.203,A -85,B 0,C 180,E1 -1761.924,E2 -1761.924} C_VEL
LIN {X 0,Y 580.254,Z 155.207,A -85,B 0,C 180,E1 -1764.452,E2 -1764.452} C_VEL
LIN {X 0,Y 580.267,Z 155.202,A -85,B 0,C 180,E1 -1766.973,E2 -1766.973} C_VEL
LIN {X 0,Y 580.285,Z 155.206,A -85,B 0,C 180,E1 -1769.424,E2 -1769.424} C_VEL
LIN {X 0,Y 580.295,Z 155.198,A -85,B 0,C 180,E1 -1772.133,E2 -1772.133} C_VEL
LIN {X 0,Y 580.288,Z 155.202,A -85,B 0,C 180,E1 -1774.919,E2 -1774.919} C_VEL
LIN {X 0,Y 580.317,Z 155.195,A -85,B 0,C 180,E1 -1777.198,E2 -1777.198} C_VEL
LIN {X 0,Y 580.272,Z 155.204,A -85,B 0,C 180,E1 -1780.176,E2 -1780.176} C_VEL
LIN {X 0,Y 580.31,Z 155.2,A -85,B 0,C 180,E1 -1783.102,E2 -1783.102} C_VEL
LIN {X 0,Y 580.303,Z 155.197,A -85,B 0,C 180,E1 -1785.982,E2 -1785.982} C_VEL
LIN {X 0,Y 580.349,Z 155.195,A -85,B 0,C 180,E1 -1788.828,E2 -1788.828} C_VEL
LIN {X 0,Y 580.314,Z 155.197,A -85,B 0,C 180,E1 -1791.643,E2 -1791.643} C_VEL
LIN {X 0,Y 580.288,Z 155.205,A -85,B 0,C 180,E1 -1793.742,E2 -1793.742} C_VEL
LIN {X 0,Y 580.248,Z 155.208,A -85,B 0,C 180,E1 -1795.832,E2 -1795.832} C_VEL
LIN {X 0,Y 580.291,Z 155.199,A -85,B 0,C 180,E1 -1797.918,E2 -1797.918} C_VEL
LIN {X 0,Y 580.341,Z 155.199,A -85,B 0,C 180,E1 -1800.694,E2 -1800.694} C_VEL
LIN {X 0,Y 580.265,Z 155.202,A -85,B 0,C 180,E1 -1803.472,E2 -1803.472} C_VEL
LIN {X 0,Y 580.314,Z 155.197,A -85,B 0,C 180,E1 -1805.56,E2 -1805.56} C_VEL
LIN {X 0,Y 580.313,Z 155.196,A -85,B 0,C 180,E1 -1808.356,E2 -1808.356} C_VEL
LIN {X 0,Y 580.341,Z 155.199,A -85,B 0,C 180,E1 -1811.234,E2 -1811.234} C_VEL
LIN {X 0,Y 580.285,Z 155.201,A -85,B 0,C 180,E1 -1814.345,E2 -1814.345} C_VEL
LIN {X 0,Y 580.28,Z 155.202,A -85,B 0,C 180,E1 -1816.918,E2 -1816.918} C_VEL
LIN {X 0,Y 580.277,Z 155.206,A -85,B 0,C 180,E1 -1819.823,E2 -1819.823} C_VEL
LIN {X 0,Y 580.317,Z 155.196,A -85,B 0,C 180,E1 -1822.801,E2 -1822.801} C_VEL
LIN {X 0,Y 580.29,Z 155.204,A -85,B 0,C 180,E1 -1825.08,E2 -1825.08} C_VEL
LIN {X 0,Y 580.293,Z 155.198,A -85,B 0,C 180,E1 -1827.866,E2 -1827.866} C_VEL
LIN {X 0,Y 580.27,Z 155.205,A -85,B 0,C 180,E1 -1830.7,E2 -1830.7} C_VEL
LIN {X 0,Y 580.273,Z 155.201,A -85,B 0,C 180,E1 -1833.319,E2 -1833.319} C_VEL
LIN {X 0,Y 580.264,Z 155.202,A -85,B 0,C 180,E1 -1836.404,E2 -1836.404} C_VEL
LIN {X 0,Y 580.29,Z 155.205,A -85,B 0,C 180,E1 -1839.19,E2 -1839.19} C_VEL
LIN {X 0,Y 580.298,Z 155.197,A -85,B 0,C 180,E1 -1841.767,E2 -1841.767} C_VEL
LIN {X 0,Y 580.246,Z 155.208,A -85,B 0,C 180,E1 -1844.628,E2 -1844.628} C_VEL
LIN {X 0,Y 580.291,Z 155.203,A -85,B 0,C 180,E1 -1847.628,E2 -1847.628} C_VEL
LIN {X 0,Y 580.264,Z 155.204,A -85,B 0,C 180,E1 -1850.069,E2 -1850.069} C_VEL
LIN {X 0,Y 580.281,Z 155.207,A -85,B 0,C 180,E1 -1853.068,E2 -1853.068} C_VEL
LIN {X 0,Y 580.295,Z 155.391,A -85,B 0,C 180,E1 -1853.943,E2 -1853.943} C_VEL
LIN {X 0,Y 580.514,Z 159.15,A -85,B 0,C 180,E1 -1855.411,E2 -1855.411} C_VEL
LIN {X 0,Y 580.44,Z 165.924,A -85,B 0,C 180,E1 -1857.948,E2 -1857.948} C_VEL
LIN {X 0,Y 580.411,Z 173.488,A -85,B 0,C 180,E1 -1860.671,E2 -1860.671} C_VEL
LIN {X 0,Y 580.346,Z 182.046,A -85,B 0,C 180,E1 -1863.656,E2 -1863.656} C_VEL
LIN {X 0,Y 580.289,Z 190.276,A -85,B 0,C 180,E1 -1866.445,E2 -1866.445} C_VEL
LIN {X 0,Y 580.23,Z 199.245,A -85,B 0,C 180,E1 -1869.438,E2 -1869.438} C_VEL
LIN {X 0,Y 580.195,Z 208.149,A -85,B 0,C 180,E1 -1872.374,E2 -1872.374} C_VEL
LIN {X 0,Y 580.135,Z 217.053,A -85,B 0,C 180,E1 -1875.263,E2 -1875.263} C_VEL
LIN {X 0,Y 580.093,Z 224.496,A -85,B 0,C 180,E1 -1877.65,E2 -1877.65} C_VEL
LIN {X 0,Y 580.798,Z 230.441,A -85,B 0,C 180,E1 -1877.776,E2 -1877.776} C_VEL
LIN {X 0,Y 580.724,Z 242.545,A -85,B 0,C 180,E1 -1878.084,E2 -1878.084} C_VEL
LIN {X 0,Y 580.606,Z 254.347,A -85,B 0,C 180,E1 -1878.516,E2 -1878.516} C_VEL
LIN {X 0,Y 580.498,Z 266.233,A -85,B 0,C 180,E1 -1879.097,E2 -1879.097} C_VEL
LIN {X 0,Y 580.439,Z 277.499,A -85,B 0,C 180,E1 -1879.801,E2 -1879.801} C_VEL
LIN {X 0,Y 580.352,Z 287.66,A -85,B 0,C 180,E1 -1880.592,E2 -1880.592} C_VEL
LIN {X 0,Y 580.279,Z 296.797,A -85,B 0,C 180,E1 -1881.469,E2 -1881.469} C_VEL
LIN {X 0,Y 580.198,Z 305.698,A -85,B 0,C 180,E1 -1882.519,E2 -1882.519} C_VEL
LIN {X 0,Y 580.119,Z 312.467,A -85,B 0,C 180,E1 -1883.505,E2 -1883.505} C_VEL
LIN {X 0,Y 580.139,Z 317.685,A -85,B 0,C 180,E1 -1884.439,E2 -1884.439} C_VEL
LIN {X 0,Y 580.108,Z 322.375,A -85,B 0,C 180,E1 -1885.484,E2 -1885.484} C_VEL
LIN {X 0,Y 580.122,Z 325.959,A -85,B 0,C 180,E1 -1886.528,E2 -1886.528} C_VEL
LIN {X 0,Y 580.043,Z 327.81,A -85,B 0,C 180,E1 -1887.223,E2 -1887.223} C_VEL
LIN {X 0,Y 580.04,Z 329.2,A -85,B 0,C 180,E1 -1887.918,E2 -1887.918} C_VEL
LIN {X 0,Y 580.04,Z 330.785,A -85,B 0,C 180,E1 -1889.306,E2 -1889.306} C_VEL
LIN {X 0,Y 580.037,Z 331,A -85,B 0,C 180,E1 -1890,E2 -1890} C_VEL
LIN {X 0,Y 580.047,Z 330.186,A -85,B 0,C 180,E1 -1891.389,E2 -1891.389} C_VEL
LIN {X 0,Y 580.04,Z 329.199,A -85,B 0,C 180,E1 -1892.083,E2 -1892.083} C_VEL
LIN {X 0,Y 580.043,Z 327.809,A -85,B 0,C 180,E1 -1892.778,E2 -1892.778} C_VEL
LIN {X 0,Y 580.11,Z 324.895,A -85,B 0,C 180,E1 -1893.821,E2 -1893.821} C_VEL
LIN {X 0,Y 580.053,Z 320.949,A -85,B 0,C 180,E1 -1894.865,E2 -1894.865} C_VEL
LIN {X 0,Y 580.139,Z 314.877,A -85,B 0,C 180,E1 -1896.085,E2 -1896.085} C_VEL
LIN {X 0,Y 580.184,Z 308.238,A -85,B 0,C 180,E1 -1897.132,E2 -1897.132} C_VEL
LIN {X 0,Y 580.25,Z 299.991,A -85,B 0,C 180,E1 -1898.182,E2 -1898.182} C_VEL
LIN {X 0,Y 580.308,Z 291.54,A -85,B 0,C 180,E1 -1899.058,E2 -1899.058} C_VEL
LIN {X 0,Y 580.411,Z 281.101,A -85,B 0,C 180,E1 -1899.936,E2 -1899.936} C_VEL
LIN {X 0,Y 580.448,Z 270.76,A -85,B 0,C 180,E1 -1900.64,E2 -1900.64} C_VEL
LIN {X 0,Y 580.562,Z 259.596,A -85,B 0,C 180,E1 -1901.247,E2 -1901.247} C_VEL
LIN {X 0,Y 580.661,Z 247.778,A -85,B 0,C 180,E1 -1901.741,E2 -1901.741} C_VEL
LIN {X 0,Y 580.771,Z 234.365,A -85,B 0,C 180,E1 -1902.137,E2 -1902.137} C_VEL
LIN {X 0,Y 580.67,Z 228.106,A -85,B 0,C 180,E1 -1902.272,E2 -1902.272} C_VEL
LIN {X 0,Y 580.094,Z 224.493,A -85,B 0,C 180,E1 -1902.351,E2 -1902.351} C_VEL
LIN {X 0,Y 580.15,Z 215.937,A -85,B 0,C 180,E1 -1905.096,E2 -1905.096} C_VEL
LIN {X 0,Y 580.191,Z 207.033,A -85,B 0,C 180,E1 -1907.991,E2 -1907.991} C_VEL
LIN {X 0,Y 580.231,Z 199.242,A -85,B 0,C 180,E1 -1910.563,E2 -1910.563} C_VEL
LIN {X 0,Y 580.291,Z 190.272,A -85,B 0,C 180,E1 -1913.556,E2 -1913.556} C_VEL
LIN {X 0,Y 580.33,Z 182.03,A -85,B 0,C 180,E1 -1916.341,E2 -1916.341} C_VEL
LIN {X 0,Y 580.358,Z 174.483,A -85,B 0,C 180,E1 -1918.971,E2 -1918.971} C_VEL
LIN {X 0,Y 580.43,Z 167.773,A -85,B 0,C 180,E1 -1921.374,E2 -1921.374} C_VEL
LIN {X 0,Y 580.485,Z 161.134,A -85,B 0,C 180,E1 -1923.841,E2 -1923.841} C_VEL
LIN {X 0,Y 580.422,Z 156.125,A -85,B 0,C 180,E1 -1925.78,E2 -1925.78} C_VEL
LIN {X 0,Y 580.253,Z 155.21,A -85,B 0,C 180,E1 -1926.232,E2 -1926.232} C_VEL
LIN {X 0,Y 580.277,Z 155.203,A -85,B 0,C 180,E1 -1929.183,E2 -1929.183} C_VEL
LIN {X 0,Y 580.301,Z 155.203,A -85,B 0,C 180,E1 -1931.764,E2 -1931.764} C_VEL
LIN {X 0,Y 580.253,Z 155.204,A -85,B 0,C 180,E1 -1934.624,E2 -1934.624} C_VEL
LIN {X 0,Y 580.264,Z 155.205,A -85,B 0,C 180,E1 -1937.292,E2 -1937.292} C_VEL
LIN {X 0,Y 580.273,Z 155.205,A -85,B 0,C 180,E1 -1940.065,E2 -1940.065} C_VEL
LIN {X 0,Y 580.28,Z 155.201,A -85,B 0,C 180,E1 -1943.063,E2 -1943.063} C_VEL
LIN {X 0,Y 580.289,Z 155.205,A -85,B 0,C 180,E1 -1945.438,E2 -1945.438} C_VEL
LIN {X 0,Y 580.29,Z 155.199,A -85,B 0,C 180,E1 -1947.966,E2 -1947.966} C_VEL
LIN {X 0,Y 580.282,Z 155.203,A -85,B 0,C 180,E1 -1950.687,E2 -1950.687} C_VEL
LIN {X 0,Y 580.247,Z 155.207,A -85,B 0,C 180,E1 -1953.375,E2 -1953.375} C_VEL
LIN {X 0,Y 580.277,Z 155.204,A -85,B 0,C 180,E1 -1955.683,E2 -1955.683} C_VEL
LIN {X 0,Y 580.275,Z 155.2,A -85,B 0,C 180,E1 -1957.948,E2 -1957.948} C_VEL
LIN {X 0,Y 580.306,Z 155.199,A -85,B 0,C 180,E1 -1960.914,E2 -1960.914} C_VEL
LIN {X 0,Y 580.264,Z 155.209,A -85,B 0,C 180,E1 -1963.825,E2 -1963.825} C_VEL
LIN {X 0,Y 580.248,Z 155.205,A -85,B 0,C 180,E1 -1966.695,E2 -1966.695} C_VEL
LIN {X 0,Y 580.358,Z 155.197,A -85,B 0,C 180,E1 -1968.828,E2 -1968.828} C_VEL
LIN {X 0,Y 580.337,Z 155.199,A -85,B 0,C 180,E1 -1972.345,E2 -1972.345} C_VEL
LIN {X 0,Y 580.328,Z 155.196,A -85,B 0,C 180,E1 -1975.137,E2 -1975.137} C_VEL
LIN {X 0,Y 580.296,Z 155.199,A -85,B 0,C 180,E1 -1977.918,E2 -1977.918} C_VEL
LIN {X 0,Y 580.349,Z 155.198,A -85,B 0,C 180,E1 -1980.694,E2 -1980.694} C_VEL
LIN {X 0,Y 580.274,Z 155.201,A -85,B 0,C 180,E1 -1983.472,E2 -1983.472} C_VEL
LIN {X 0,Y 580.32,Z 155.2,A -85,B 0,C 180,E1 -1985.56,E2 -1985.56} C_VEL
LIN {X 0,Y 580.311,Z 155.197,A -85,B 0,C 180,E1 -1988.357,E2 -1988.357} C_VEL
LIN {X 0,Y 580.301,Z 155.2,A -85,B 0,C 180,E1 -1991.209,E2 -1991.209} C_VEL
LIN {X 0,Y 580.295,Z 155.202,A -85,B 0,C 180,E1 -1994.345,E2 -1994.345} C_VEL
LIN {X 0,Y 580.314,Z 155.196,A -85,B 0,C 180,E1 -1996.926,E2 -1996.926} C_VEL
LIN {X 0,Y 580.292,Z 155.199,A -85,B 0,C 180,E1 -1999.823,E2 -1999.823} C_VEL
LIN {X 0,Y 580.263,Z 155.204,A -85,B 0,C 180,E1 -2001.36,E2 -2001.36} C_VEL
LIN {X 0,Y 579.573,Z 155.29,A -85,B 0,C 180,E1 -2001.94,E2 -2001.94} C_VEL
LIN {X 0,Y 576.695,Z 155.65,A -85,B 0,C 180,E1 -2002.879,E2 -2002.879} C_VEL
LIN {X 0,Y 574.294,Z 155.948,A -85,B 0,C 180,E1 -2003.636,E2 -2003.636} C_VEL
LIN {X 0,Y 573.293,Z 156.077,A -85,B 0,C 180,E1 -2004.22,E2 -2004.22} C_VEL
LIN {X 0,Y 573.226,Z 156.08,A -85,B 0,C 180,E1 -2004.417,E2 -2004.417} C_VEL
LIN {X 0,Y 573.242,Z 156.077,A -85,B 0,C 180,E1 -2006.977,E2 -2006.977} C_VEL
LIN {X 0,Y 573.234,Z 156.082,A -85,B 0,C 180,E1 -2009.492,E2 -2009.492} C_VEL
LIN {X 0,Y 573.24,Z 156.079,A -85,B 0,C 180,E1 -2012.232,E2 -2012.232} C_VEL
LIN {X 0,Y 573.22,Z 156.082,A -85,B 0,C 180,E1 -2014.774,E2 -2014.774} C_VEL
LIN {X 0,Y 573.214,Z 156.086,A -85,B 0,C 180,E1 -2017.81,E2 -2017.81} C_VEL
LIN {X 0,Y 573.253,Z 156.076,A -85,B 0,C 180,E1 -2020.53,E2 -2020.53} C_VEL
LIN {X 0,Y 573.239,Z 156.077,A -85,B 0,C 180,E1 -2023.672,E2 -2023.672} C_VEL
LIN {X 0,Y 573.228,Z 156.08,A -85,B 0,C 180,E1 -2026.643,E2 -2026.643} C_VEL
LIN {X 0,Y 573.234,Z 156.084,A -85,B 0,C 180,E1 -2029.477,E2 -2029.477} C_VEL
LIN {X 0,Y 573.198,Z 156.083,A -85,B 0,C 180,E1 -2032.192,E2 -2032.192} C_VEL
LIN {X 0,Y 573.182,Z 156.33,A -85,B 0,C 180,E1 -2032.844,E2 -2032.844} C_VEL
LIN {X 0,Y 573.148,Z 160.977,A -85,B 0,C 180,E1 -2035.665,E2 -2035.665} C_VEL
LIN {X 0,Y 573.156,Z 165.175,A -85,B 0,C 180,E1 -2038.181,E2 -2038.181} C_VEL
LIN {X 0,Y 573.126,Z 169.328,A -85,B 0,C 180,E1 -2040.628,E2 -2040.628} C_VEL
LIN {X 0,Y 573.077,Z 173.47,A -85,B 0,C 180,E1 -2043.017,E2 -2043.017} C_VEL
LIN {X 0,Y 573.073,Z 177.57,A -85,B 0,C 180,E1 -2045.358,E2 -2045.358} C_VEL
LIN {X 0,Y 573.026,Z 183.023,A -85,B 0,C 180,E1 -2048.412,E2 -2048.412} C_VEL
LIN {X 0,Y 573.006,Z 188.617,A -85,B 0,C 180,E1 -2051.405,E2 -2051.405} C_VEL
LIN {X 0,Y 572.962,Z 192.807,A -85,B 0,C 180,E1 -2053.614,E2 -2053.614} C_VEL
LIN {X 0,Y 572.942,Z 196.634,A -85,B 0,C 180,E1 -2055.576,E2 -2055.576} C_VEL
LIN {X 0,Y 573.856,Z 203.752,A -85,B 0,C 180,E1 -2055.744,E2 -2055.744} C_VEL
LIN {X 0,Y 573.747,Z 217.06,A -85,B 0,C 180,E1 -2056.136,E2 -2056.136} C_VEL
LIN {X 0,Y 573.611,Z 228.98,A -85,B 0,C 180,E1 -2056.629,E2 -2056.629} C_VEL
LIN {X 0,Y 573.424,Z 240.479,A -85,B 0,C 180,E1 -2057.255,E2 -2057.255} C_VEL
LIN {X 0,Y 573.38,Z 252.107,A -85,B 0,C 180,E1 -2058.063,E2 -2058.063} C_VEL
LIN {X 0,Y 573.26,Z 261.777,A -85,B 0,C 180,E1 -2058.897,E2 -2058.897} C_VEL
LIN {X 0,Y 573.199,Z 271.467,A -85,B 0,C 180,E1 -2059.938,E2 -2059.938} C_VEL
LIN {X 0,Y 573.11,Z 279.495,A -85,B 0,C 180,E1 -2061.005,E2 -2061.005} C_VEL
LIN {X 0,Y 573.06,Z 284.92,A -85,B 0,C 180,E1 -2061.892,E2 -2061.892} C_VEL
LIN {X 0,Y 573.051,Z 290.225,A -85,B 0,C 180,E1 -2062.955,E2 -2062.955} C_VEL
LIN {X 0,Y 573.012,Z 294.349,A -85,B 0,C 180,E1 -2064.016,E2 -2064.016} C_VEL
LIN {X 0,Y 572.944,Z 297.415,A -85,B 0,C 180,E1 -2065.074,E2 -2065.074} C_VEL
LIN {X 0,Y 573.009,Z 298.937,A -85,B 0,C 180,E1 -2065.78,E2 -2065.78} C_VEL
LIN {X 0,Y 573.007,Z 300.009,A -85,B 0,C 180,E1 -2066.484,E2 -2066.484} C_VEL
LIN {X 0,Y 572.938,Z 300.972,A -85,B 0,C 180,E1 -2067.891,E2 -2067.891} C_VEL
LIN {X 0,Y 572.946,Z 300.879,A -85,B 0,C 180,E1 -2068.594,E2 -2068.594} C_VEL
LIN {X 0,Y 572.941,Z 299.444,A -85,B 0,C 180,E1 -2070,E2 -2070} C_VEL
LIN {X 0,Y 572.942,Z 298.136,A -85,B 0,C 180,E1 -2070.702,E2 -2070.702} C_VEL
LIN {X 0,Y 572.995,Z 295.368,A -85,B 0,C 180,E1 -2071.757,E2 -2071.757} C_VEL
LIN {X 0,Y 572.982,Z 291.591,A -85,B 0,C 180,E1 -2072.812,E2 -2072.812} C_VEL
LIN {X 0,Y 573.071,Z 286.698,A -85,B 0,C 180,E1 -2073.867,E2 -2073.867} C_VEL
LIN {X 0,Y 573.125,Z 280.547,A -85,B 0,C 180,E1 -2074.923,E2 -2074.923} C_VEL
LIN {X 0,Y 573.157,Z 272.898,A -85,B 0,C 180,E1 -2075.982,E2 -2075.982} C_VEL
LIN {X 0,Y 573.248,Z 264.794,A -85,B 0,C 180,E1 -2076.892,E2 -2076.892} C_VEL
LIN {X 0,Y 573.348,Z 254.479,A -85,B 0,C 180,E1 -2077.837,E2 -2077.837} C_VEL
LIN {X 0,Y 573.448,Z 243.661,A -85,B 0,C 180,E1 -2078.633,E2 -2078.633} C_VEL
LIN {X 0,Y 573.53,Z 233.094,A -85,B 0,C 180,E1 -2079.254,E2 -2079.254} C_VEL
LIN {X 0,Y 573.687,Z 220.402,A -85,B 0,C 180,E1 -2079.83,E2 -2079.83} C_VEL
LIN {X 0,Y 573.804,Z 207.626,A -85,B 0,C 180,E1 -2080.251,E2 -2080.251} C_VEL
LIN {X 0,Y 573.69,Z 201.15,A -85,B 0,C 180,E1 -2080.409,E2 -2080.409} C_VEL
LIN {X 0,Y 572.945,Z 196.523,A -85,B 0,C 180,E1 -2080.534,E2 -2080.534} C_VEL
LIN {X 0,Y 572.972,Z 192.278,A -85,B 0,C 180,E1 -2082.754,E2 -2082.754} C_VEL
LIN {X 0,Y 573.031,Z 188.167,A -85,B 0,C 180,E1 -2084.924,E2 -2084.924} C_VEL
LIN {X 0,Y 573.043,Z 182.707,A -85,B 0,C 180,E1 -2087.853,E2 -2087.853} C_VEL
LIN {X 0,Y 573.022,Z 178.709,A -85,B 0,C 180,E1 -2090.083,E2 -2090.083} C_VEL
LIN {X 0,Y 573.088,Z 174.733,A -85,B 0,C 180,E1 -2092.342,E2 -2092.342} C_VEL
LIN {X 0,Y 573.137,Z 170.401,A -85,B 0,C 180,E1 -2094.849,E2 -2094.849} C_VEL
LIN {X 0,Y 573.156,Z 165.404,A -85,B 0,C 180,E1 -2097.769,E2 -2097.769} C_VEL
LIN {X 0,Y 573.163,Z 161.368,A -85,B 0,C 180,E1 -2100.178,E2 -2100.178} C_VEL
LIN {X 0,Y 573.162,Z 157.261,A -85,B 0,C 180,E1 -2102.648,E2 -2102.648} C_VEL
LIN {X 0,Y 573.166,Z 156.091,A -85,B 0,C 180,E1 -2103.508,E2 -2103.508} C_VEL
LIN {X 0,Y 573.179,Z 156.085,A -85,B 0,C 180,E1 -2106.05,E2 -2106.05} C_VEL
LIN {X 0,Y 573.225,Z 156.084,A -85,B 0,C 180,E1 -2108.699,E2 -2108.699} C_VEL
LIN {X 0,Y 573.237,Z 156.08,A -85,B 0,C 180,E1 -2111.593,E2 -2111.593} C_VEL
LIN {X 0,Y 573.22,Z 156.08,A -85,B 0,C 180,E1 -2114.33,E2 -2114.33} C_VEL
LIN {X 0,Y 573.24,Z 156.082,A -85,B 0,C 180,E1 -2117.353,E2 -2117.353} C_VEL
LIN {X 0,Y 573.226,Z 156.082,A -85,B 0,C 180,E1 -2120.391,E2 -2120.391} C_VEL
LIN {X 0,Y 573.225,Z 156.079,A -85,B 0,C 180,E1 -2123.075,E2 -2123.075} C_VEL
LIN {X 0,Y 573.239,Z 156.081,A -85,B 0,C 180,E1 -2125.669,E2 -2125.669} C_VEL
LIN {X 0,Y 573.227,Z 156.08,A -85,B 0,C 180,E1 -2128.183,E2 -2128.183} C_VEL
LIN {X 0,Y 573.258,Z 156.076,A -85,B 0,C 180,E1 -2130.633,E2 -2130.633} C_VEL
LIN {X 0,Y 573.249,Z 156.076,A -85,B 0,C 180,E1 -2133.496,E2 -2133.496} C_VEL
LIN {X 0,Y 573.242,Z 156.08,A -85,B 0,C 180,E1 -2136.135,E2 -2136.135} C_VEL
LIN {X 0,Y 573.225,Z 156.079,A -85,B 0,C 180,E1 -2138.704,E2 -2138.704} C_VEL
LIN {X 0,Y 573.192,Z 156.088,A -85,B 0,C 180,E1 -2141.41,E2 -2141.41} C_VEL
LIN {X 0,Y 573.239,Z 156.081,A -85,B 0,C 180,E1 -2143.621,E2 -2143.621} C_VEL
LIN {X 0,Y 573.23,Z 156.082,A -85,B 0,C 180,E1 -2146.529,E2 -2146.529} C_VEL
LIN {X 0,Y 573.274,Z 156.072,A -85,B 0,C 180,E1 -2149.403,E2 -2149.403} C_VEL
LIN {X 0,Y 573.278,Z 156.077,A -85,B 0,C 180,E1 -2152.25,E2 -2152.25} C_VEL
LIN {X 0,Y 573.293,Z 156.071,A -85,B 0,C 180,E1 -2155.077,E2 -2155.077} C_VEL
LIN {X 0,Y 573.263,Z 156.075,A -85,B 0,C 180,E1 -2157.892,E2 -2157.892} C_VEL
LIN {X 0,Y 573.309,Z 156.075,A -85,B 0,C 180,E1 -2160.702,E2 -2160.702} C_VEL
LIN {X 0,Y 573.217,Z 156.08,A -85,B 0,C 180,E1 -2163.514,E2 -2163.514} C_VEL
LIN {X 0,Y 573.282,Z 156.074,A -85,B 0,C 180,E1 -2165.628,E2 -2165.628} C_VEL
LIN {X 0,Y 573.283,Z 156.071,A -85,B 0,C 180,E1 -2168.459,E2 -2168.459} C_VEL
LIN {X 0,Y 573.285,Z 156.078,A -85,B 0,C 180,E1 -2171.312,E2 -2171.312} C_VEL
LIN {X 0,Y 573.249,Z 156.079,A -85,B 0,C 180,E1 -2174.429,E2 -2174.429} C_VEL
LIN {X 0,Y 573.223,Z 156.08,A -85,B 0,C 180,E1 -2177.113,E2 -2177.113} C_VEL
LIN {X 0,Y 573.227,Z 156.085,A -85,B 0,C 180,E1 -2180.077,E2 -2180.077} C_VEL
LIN {X 0,Y 573.273,Z 156.076,A -85,B 0,C 180,E1 -2183.164,E2 -2183.164} C_VEL
LIN {X 0,Y 573.264,Z 156.073,A -85,B 0,C 180,E1 -2186.19,E2 -2186.19} C_VEL
LIN {X 0,Y 573.244,Z 156.082,A -85,B 0,C 180,E1 -2188.564,E2 -2188.564} C_VEL
LIN {X 0,Y 573.211,Z 156.081,A -85,B 0,C 180,E1 -2190.994,E2 -2190.994} C_VEL
LIN {X 0,Y 573.231,Z 156.08,A -85,B 0,C 180,E1 -2193.526,E2 -2193.526} C_VEL
LIN {X 0,Y 573.228,Z 156.081,A -85,B 0,C 180,E1 -2196.051,E2 -2196.051} C_VEL
LIN {X 0,Y 573.228,Z 156.08,A -85,B 0,C 180,E1 -2198.703,E2 -2198.703} C_VEL
LIN {X 0,Y 573.244,Z 156.076,A -85,B 0,C 180,E1 -2201.6,E2 -2201.6} C_VEL
LIN {X 0,Y 573.217,Z 156.087,A -85,B 0,C 180,E1 -2204.335,E2 -2204.335} C_VEL
LIN {X 0,Y 573.241,Z 156.079,A -85,B 0,C 180,E1 -2207.359,E2 -2207.359} C_VEL
LIN {X 0,Y 573.256,Z 156.082,A -85,B 0,C 180,E1 -2209.48,E2 -2209.48} C_VEL
LIN {X 0,Y 573.213,Z 156.082,A -85,B 0,C 180,E1 -2212.195,E2 -2212.195} C_VEL
LIN {X 0,Y 573.223,Z 156.114,A -85,B 0,C 180,E1 -2213.735,E2 -2213.735} C_VEL
LIN {X 0,Y 573.517,Z 159.767,A -85,B 0,C 180,E1 -2215.188,E2 -2215.188} C_VEL
LIN {X 0,Y 573.441,Z 166.484,A -85,B 0,C 180,E1 -2217.742,E2 -2217.742} C_VEL
LIN {X 0,Y 573.408,Z 174.429,A -85,B 0,C 180,E1 -2220.645,E2 -2220.645} C_VEL
LIN {X 0,Y 573.302,Z 183.408,A -85,B 0,C 180,E1 -2223.815,E2 -2223.815} C_VEL
LIN {X 0,Y 573.238,Z 191.313,A -85,B 0,C 180,E1 -2226.521,E2 -2226.521} C_VEL
LIN {X 0,Y 573.175,Z 199.226,A -85,B 0,C 180,E1 -2229.173,E2 -2229.173} C_VEL
LIN {X 0,Y 573.123,Z 207.036,A -85,B 0,C 180,E1 -2231.78,E2 -2231.78} C_VEL
LIN {X 0,Y 573.097,Z 214.827,A -85,B 0,C 180,E1 -2234.35,E2 -2234.35} C_VEL
LIN {X 0,Y 573.058,Z 222.618,A -85,B 0,C 180,E1 -2236.888,E2 -2236.888} C_VEL
LIN {X 0,Y 573.028,Z 224.496,A -85,B 0,C 180,E1 -2237.495,E2 -2237.495} C_VEL
LIN {X 0,Y 573.866,Z 230.44,A -85,B 0,C 180,E1 -2237.626,E2 -2237.626} C_VEL
LIN {X 0,Y 573.784,Z 242.546,A -85,B 0,C 180,E1 -2237.938,E2 -2237.938} C_VEL
LIN {X 0,Y 573.646,Z 254.345,A -85,B 0,C 180,E1 -2238.375,E2 -2238.375} C_VEL
LIN {X 0,Y 573.516,Z 266.701,A -85,B 0,C 180,E1 -2238.989,E2 -2238.989} C_VEL
LIN {X 0,Y 573.433,Z 277.5,A -85,B 0,C 180,E1 -2239.676,E2 -2239.676} C_VEL
LIN {X 0,Y 573.307,Z 287.66,A -85,B 0,C 180,E1 -2240.475,E2 -2240.475} C_VEL
LIN {X 0,Y 573.214,Z 296.797,A -85,B 0,C 180,E1 -2241.363,E2 -2241.363} C_VEL
LIN {X 0,Y 573.141,Z 305.697,A -85,B 0,C 180,E1 -2242.426,E2 -2242.426} C_VEL
LIN {X 0,Y 573.05,Z 312.407,A -85,B 0,C 180,E1 -2243.415,E2 -2243.415} C_VEL
LIN {X 0,Y 573.07,Z 317.684,A -85,B 0,C 180,E1 -2244.371,E2 -2244.371} C_VEL
LIN {X 0,Y 573.028,Z 322.375,A -85,B 0,C 180,E1 -2245.428,E2 -2245.428} C_VEL
LIN {X 0,Y 573.022,Z 325.96,A -85,B 0,C 180,E1 -2246.485,E2 -2246.485} C_VEL
LIN {X 0,Y 572.959,Z 327.81,A -85,B 0,C 180,E1 -2247.188,E2 -2247.188} C_VEL
LIN {X 0,Y 572.94,Z 329.199,A -85,B 0,C 180,E1 -2247.892,E2 -2247.892} C_VEL
LIN {X 0,Y 572.941,Z 330.785,A -85,B 0,C 180,E1 -2249.298,E2 -2249.298} C_VEL
LIN {X 0,Y 572.938,Z 331,A -85,B 0,C 180,E1 -2250,E2 -2250} C_VEL
LIN {X 0,Y 572.946,Z 330.186,A -85,B 0,C 180,E1 -2251.406,E2 -2251.406} C_VEL
LIN {X 0,Y 572.94,Z 329.199,A -85,B 0,C 180,E1 -2252.109,E2 -2252.109} C_VEL
LIN {X 0,Y 572.959,Z 327.809,A -85,B 0,C 180,E1 -2252.813,E2 -2252.813} C_VEL
LIN {X 0,Y 573.015,Z 324.895,A -85,B 0,C 180,E1 -2253.868,E2 -2253.868} C_VEL
LIN {X 0,Y 572.963,Z 320.948,A -85,B 0,C 180,E1 -2254.926,E2 -2254.926} C_VEL
LIN {X 0,Y 573.065,Z 314.876,A -85,B 0,C 180,E1 -2256.16,E2 -2256.16} C_VEL
LIN {X 0,Y 573.119,Z 308.238,A -85,B 0,C 180,E1 -2257.221,E2 -2257.221} C_VEL
LIN {X 0,Y 573.201,Z 299.992,A -85,B 0,C 180,E1 -2258.283,E2 -2258.283} C_VEL
LIN {X 0,Y 573.287,Z 291.541,A -85,B 0,C 180,E1 -2259.17,E2 -2259.17} C_VEL
LIN {X 0,Y 573.411,Z 281.101,A -85,B 0,C 180,E1 -2260.058,E2 -2260.058} C_VEL
LIN {X 0,Y 573.515,Z 269.543,A -85,B 0,C 180,E1 -2260.847,E2 -2260.847} C_VEL
LIN {X 0,Y 573.608,Z 257.892,A -85,B 0,C 180,E1 -2261.466,E2 -2261.466} C_VEL
LIN {X 0,Y 573.758,Z 245.182,A -85,B 0,C 180,E1 -2261.974,E2 -2261.974} C_VEL
LIN {X 0,Y 573.847,Z 232.535,A -85,B 0,C 180,E1 -2262.331,E2 -2262.331} C_VEL
LIN {X 0,Y 573.667,Z 228.669,A -85,B 0,C 180,E1 -2262.413,E2 -2262.413} C_VEL
LIN {X 0,Y 573.028,Z 224.493,A -85,B 0,C 180,E1 -2262.506,E2 -2262.506} C_VEL
LIN {X 0,Y 573.079,Z 215.937,A -85,B 0,C 180,E1 -2265.287,E2 -2265.287} C_VEL
LIN {X 0,Y 573.134,Z 208.146,A -85,B 0,C 180,E1 -2267.851,E2 -2267.851} C_VEL
LIN {X 0,Y 573.185,Z 200.353,A -85,B 0,C 180,E1 -2270.452,E2 -2270.452} C_VEL
LIN {X 0,Y 573.209,Z 192.325,A -85,B 0,C 180,E1 -2273.138,E2 -2273.138} C_VEL
LIN {X 0,Y 573.273,Z 184.513,A -85,B 0,C 180,E1 -2275.797,E2 -2275.797} C_VEL
LIN {X 0,Y 573.349,Z 176.658,A -85,B 0,C 180,E1 -2278.557,E2 -2278.557} C_VEL
LIN {X 0,Y 573.421,Z 168.815,A -85,B 0,C 180,E1 -2281.39,E2 -2281.39} C_VEL
LIN {X 0,Y 573.489,Z 163.047,A -85,B 0,C 180,E1 -2283.558,E2 -2283.558} C_VEL
LIN {X 0,Y 573.516,Z 157.887,A -85,B 0,C 180,E1 -2285.574,E2 -2285.574} C_VEL
LIN {X 0,Y 573.227,Z 156.085,A -85,B 0,C 180,E1 -2286.375,E2 -2286.375} C_VEL
LIN {X 0,Y 573.228,Z 156.081,A -85,B 0,C 180,E1 -2289.43,E2 -2289.43} C_VEL
LIN {X 0,Y 573.241,Z 156.081,A -85,B 0,C 180,E1 -2291.594,E2 -2291.594} C_VEL
LIN {X 0,Y 573.224,Z 156.079,A -85,B 0,C 180,E1 -2294.331,E2 -2294.331} C_VEL
LIN {X 0,Y 573.226,Z 156.081,A -85,B 0,C 180,E1 -2297.356,E2 -2297.356} C_VEL
LIN {X 0,Y 573.229,Z 156.082,A -85,B 0,C 180,E1 -2300.566,E2 -2300.566} C_VEL
LIN {X 0,Y 573.235,Z 156.078,A -85,B 0,C 180,E1 -2303.076,E2 -2303.076} C_VEL
LIN {X 0,Y 573.258,Z 156.077,A -85,B 0,C 180,E1 -2305.671,E2 -2305.671} C_VEL
LIN {X 0,Y 573.231,Z 156.079,A -85,B 0,C 180,E1 -2308.184,E2 -2308.184} C_VEL
LIN {X 0,Y 573.246,Z 156.081,A -85,B 0,C 180,E1 -2310.633,E2 -2310.633} C_VEL
